REGION Network 36: Interface Signals 06 / Interface Signals ET200SP_204
   // Aufruf des Schnittstellen Signal Bausteins / Call the interface signals bool blocks
   RUNG wire#powerrail
      #instSignalsLeft[43](signal00 := "ET200SP_204"."SP204.00 Main OP: Emergency stop", signal01 := "ET200SP_204".SPARE1, signal02 := "ET200SP_204".SPARE2, signal03 := "ET200SP_204".SPARE3, signal04 := "ET200SP_204".RESERVED, signal05 := "ET200SP_204".SPARE4, signal06 := "ET200SP_204".SPARE5, signal07 := "ET200SP_204".SPARE6, signal08 :=, signal09 :=, signal10 :=, signal11 :=, signal12 :=, signal13 :=, signal14 :=, signal15 :=, interfaceSignals := #statInterfaceSignalsHmi[43].valueSymbolLeft)
      #instSignalsRight[43](signal00 :=, signal01 :=, signal02 :=, signal03 :=, signal04 :=, signal05 :=, signal06 :=, signal07 :=, signal08 :=, signal09 :=, signal10 :=, signal11 :=, signal12 :=, signal13 :=, signal14 :=, signal15 :=, interfaceSignals := #statInterfaceSignalsHmi[43].valueSymbolRight)
   END_RUNG
   // the same network as SCL:
   #instSignalsLeft[43](signal00 := "ET200SP_204"."SP204.00 Main OP: Emergency stop",   // "LAF_InterfaceSignalsBool"
                        signal01 := "ET200SP_204".SPARE1,
                        signal02 := "ET200SP_204".SPARE2,
                        signal03 := "ET200SP_204".SPARE3,
                        signal04 := "ET200SP_204".RESERVED,
                        signal05 := "ET200SP_204".SPARE4,
                        signal06 := "ET200SP_204".SPARE5,
                        signal07 := "ET200SP_204".SPARE6,
                        interfaceSignals := #statInterfaceSignalsHmi[43].valueSymbolLeft,
                        ENO => #_w1);
   IF #_w1 THEN
       #instSignalsRight[43](interfaceSignals := #statInterfaceSignalsHmi[43].valueSymbolRight);   // "LAF_InterfaceSignalsBool"
   END_IF;
END_REGION

REGION Network 37: Interface Signals 06 / Interface Signals ET200SP_205
   // Aufruf des Schnittstellen Signal Bausteins / Call the interface signals bool blocks
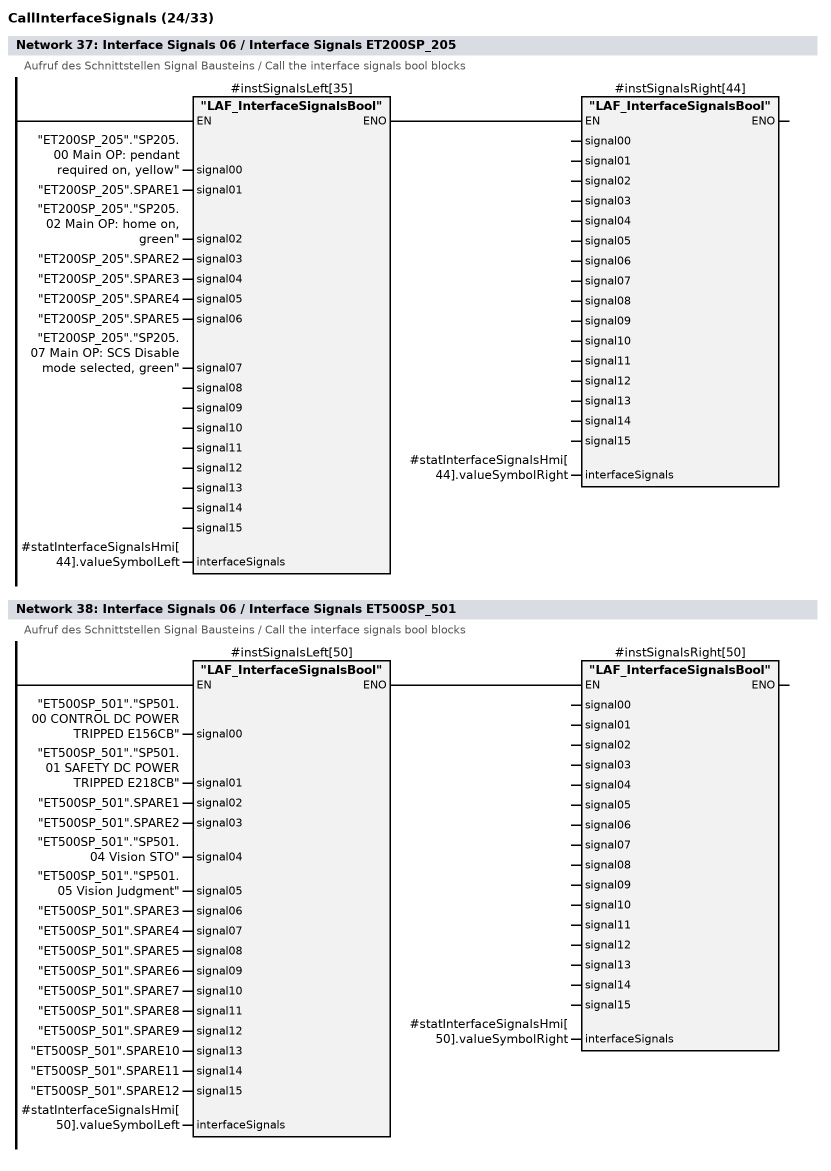
   RUNG wire#powerrail
      #instSignalsLeft[35](signal00 := "ET200SP_205"."SP205.00 Main OP: pendant required on, yellow", signal01 := "ET200SP_205".SPARE1, signal02 := "ET200SP_205"."SP205.02 Main OP: home on, green", signal03 := "ET200SP_205".SPARE2, signal04 := "ET200SP_205".SPARE3, signal05 := "ET200SP_205".SPARE4, signal06 := "ET200SP_205".SPARE5, signal07 := "ET200SP_205"."SP205.07 Main OP: SCS Disable mode selected, green", signal08 :=, signal09 :=, signal10 :=, signal11 :=, signal12 :=, signal13 :=, signal14 :=, signal15 :=, interfaceSignals := #statInterfaceSignalsHmi[44].valueSymbolLeft)
      #instSignalsRight[44](signal00 :=, signal01 :=, signal02 :=, signal03 :=, signal04 :=, signal05 :=, signal06 :=, signal07 :=, signal08 :=, signal09 :=, signal10 :=, signal11 :=, signal12 :=, signal13 :=, signal14 :=, signal15 :=, interfaceSignals := #statInterfaceSignalsHmi[44].valueSymbolRight)
   END_RUNG
   // the same network as SCL:
   #instSignalsLeft[35](signal00 := "ET200SP_205"."SP205.00 Main OP: pendant required on, yellow",   // "LAF_InterfaceSignalsBool"
                        signal01 := "ET200SP_205".SPARE1,
                        signal02 := "ET200SP_205"."SP205.02 Main OP: home on, green",
                        signal03 := "ET200SP_205".SPARE2,
                        signal04 := "ET200SP_205".SPARE3,
                        signal05 := "ET200SP_205".SPARE4,
                        signal06 := "ET200SP_205".SPARE5,
                        signal07 := "ET200SP_205"."SP205.07 Main OP: SCS Disable mode selected, green",
                        interfaceSignals := #statInterfaceSignalsHmi[44].valueSymbolLeft,
                        ENO => #_w1);
   IF #_w1 THEN
       #instSignalsRight[44](interfaceSignals := #statInterfaceSignalsHmi[44].valueSymbolRight);   // "LAF_InterfaceSignalsBool"
   END_IF;
END_REGION

REGION Network 38: Interface Signals 06 / Interface Signals ET500SP_501
   // Aufruf des Schnittstellen Signal Bausteins / Call the interface signals bool blocks
   RUNG wire#powerrail
      #instSignalsLeft[50](signal00 := "ET500SP_501"."SP501.00 CONTROL DC POWER TRIPPED E156CB", signal01 := "ET500SP_501"."SP501.01 SAFETY DC POWER TRIPPED E218CB", signal02 := "ET500SP_501".SPARE1, signal03 := "ET500SP_501".SPARE2, signal04 := "ET500SP_501"."SP501.04 Vision STO", signal05 := "ET500SP_501"."SP501.05 Vision Judgment", signal06 := "ET500SP_501".SPARE3, signal07 := "ET500SP_501".SPARE4, signal08 := "ET500SP_501".SPARE5, signal09 := "ET500SP_501".SPARE6, signal10 := "ET500SP_501".SPARE7, signal11 := "ET500SP_501".SPARE8, signal12 := "ET500SP_501".SPARE9, signal13 := "ET500SP_501".SPARE10, signal14 := "ET500SP_501".SPARE11, signal15 := "ET500SP_501".SPARE12, interfaceSignals := #statInterfaceSignalsHmi[50].valueSymbolLeft)
      #instSignalsRight[50](signal00 :=, signal01 :=, signal02 :=, signal03 :=, signal04 :=, signal05 :=, signal06 :=, signal07 :=, signal08 :=, signal09 :=, signal10 :=, signal11 :=, signal12 :=, signal13 :=, signal14 :=, signal15 :=, interfaceSignals := #statInterfaceSignalsHmi[50].valueSymbolRight)
   END_RUNG
   // the same network as SCL:
   #instSignalsLeft[50](signal00 := "ET500SP_501"."SP501.00 CONTROL DC POWER TRIPPED E156CB",   // "LAF_InterfaceSignalsBool"
                        signal01 := "ET500SP_501"."SP501.01 SAFETY DC POWER TRIPPED E218CB",
                        signal02 := "ET500SP_501".SPARE1,
                        signal03 := "ET500SP_501".SPARE2,
                        signal04 := "ET500SP_501"."SP501.04 Vision STO",
                        signal05 := "ET500SP_501"."SP501.05 Vision Judgment",
                        signal06 := "ET500SP_501".SPARE3,
                        signal07 := "ET500SP_501".SPARE4,
                        signal08 := "ET500SP_501".SPARE5,
                        signal09 := "ET500SP_501".SPARE6,
                        signal10 := "ET500SP_501".SPARE7,
                        signal11 := "ET500SP_501".SPARE8,
                        signal12 := "ET500SP_501".SPARE9,
                        signal13 := "ET500SP_501".SPARE10,
                        signal14 := "ET500SP_501".SPARE11,
                        signal15 := "ET500SP_501".SPARE12,
                        interfaceSignals := #statInterfaceSignalsHmi[50].valueSymbolLeft,
                        ENO => #_w1);
   IF #_w1 THEN
       #instSignalsRight[50](interfaceSignals := #statInterfaceSignalsHmi[50].valueSymbolRight);   // "LAF_InterfaceSignalsBool"
   END_IF;
END_REGION

REGION Network 39: Interface Signals 06 / Interface Signals ET500SP_502
   // Aufruf des Schnittstellen Signal Bausteins / Call the interface signals bool blocks
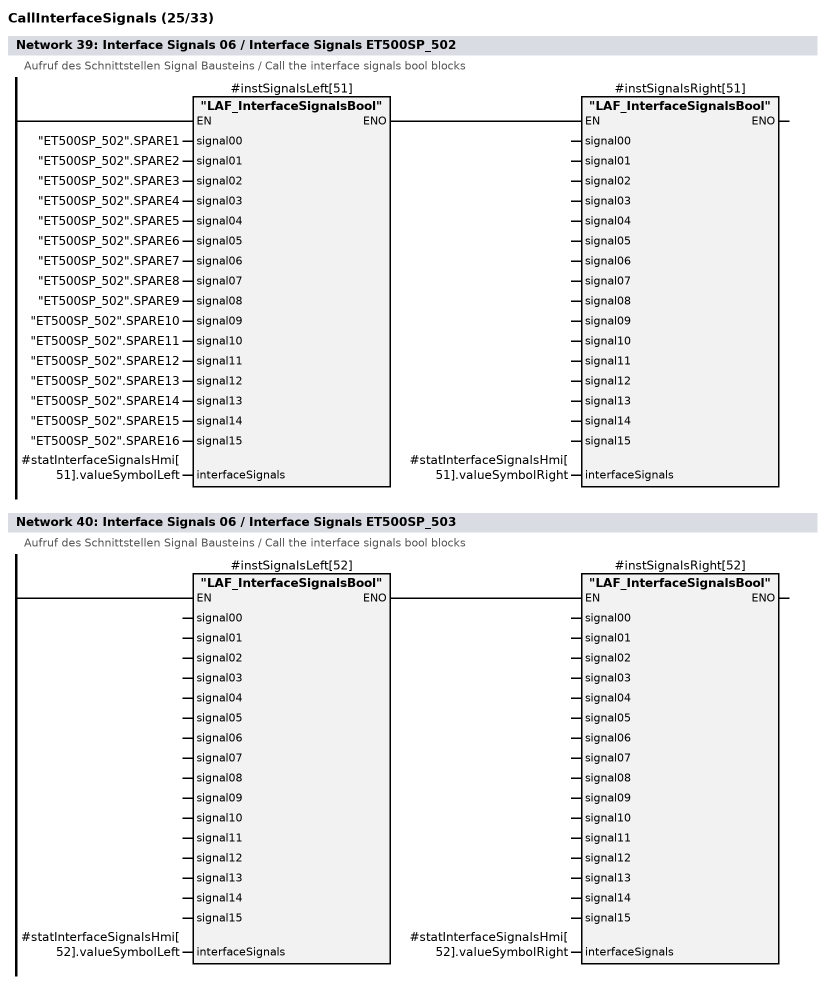
   RUNG wire#powerrail
      #instSignalsLeft[51](signal00 := "ET500SP_502".SPARE1, signal01 := "ET500SP_502".SPARE2, signal02 := "ET500SP_502".SPARE3, signal03 := "ET500SP_502".SPARE4, signal04 := "ET500SP_502".SPARE5, signal05 := "ET500SP_502".SPARE6, signal06 := "ET500SP_502".SPARE7, signal07 := "ET500SP_502".SPARE8, signal08 := "ET500SP_502".SPARE9, signal09 := "ET500SP_502".SPARE10, signal10 := "ET500SP_502".SPARE11, signal11 := "ET500SP_502".SPARE12, signal12 := "ET500SP_502".SPARE13, signal13 := "ET500SP_502".SPARE14, signal14 := "ET500SP_502".SPARE15, signal15 := "ET500SP_502".SPARE16, interfaceSignals := #statInterfaceSignalsHmi[51].valueSymbolLeft)
      #instSignalsRight[51](signal00 :=, signal01 :=, signal02 :=, signal03 :=, signal04 :=, signal05 :=, signal06 :=, signal07 :=, signal08 :=, signal09 :=, signal10 :=, signal11 :=, signal12 :=, signal13 :=, signal14 :=, signal15 :=, interfaceSignals := #statInterfaceSignalsHmi[51].valueSymbolRight)
   END_RUNG
   // the same network as SCL:
   #instSignalsLeft[51](signal00 := "ET500SP_502".SPARE1,   // "LAF_InterfaceSignalsBool"
                        signal01 := "ET500SP_502".SPARE2,
                        signal02 := "ET500SP_502".SPARE3,
                        signal03 := "ET500SP_502".SPARE4,
                        signal04 := "ET500SP_502".SPARE5,
                        signal05 := "ET500SP_502".SPARE6,
                        signal06 := "ET500SP_502".SPARE7,
                        signal07 := "ET500SP_502".SPARE8,
                        signal08 := "ET500SP_502".SPARE9,
                        signal09 := "ET500SP_502".SPARE10,
                        signal10 := "ET500SP_502".SPARE11,
                        signal11 := "ET500SP_502".SPARE12,
                        signal12 := "ET500SP_502".SPARE13,
                        signal13 := "ET500SP_502".SPARE14,
                        signal14 := "ET500SP_502".SPARE15,
                        signal15 := "ET500SP_502".SPARE16,
                        interfaceSignals := #statInterfaceSignalsHmi[51].valueSymbolLeft,
                        ENO => #_w1);
   IF #_w1 THEN
       #instSignalsRight[51](interfaceSignals := #statInterfaceSignalsHmi[51].valueSymbolRight);   // "LAF_InterfaceSignalsBool"
   END_IF;
END_REGION

REGION Network 40: Interface Signals 06 / Interface Signals ET500SP_503
   // Aufruf des Schnittstellen Signal Bausteins / Call the interface signals bool blocks
   RUNG wire#powerrail
      #instSignalsLeft[52](signal00 :=, signal01 :=, signal02 :=, signal03 :=, signal04 :=, signal05 :=, signal06 :=, signal07 :=, signal08 :=, signal09 :=, signal10 :=, signal11 :=, signal12 :=, signal13 :=, signal14 :=, signal15 :=, interfaceSignals := #statInterfaceSignalsHmi[52].valueSymbolLeft)
      #instSignalsRight[52](signal00 :=, signal01 :=, signal02 :=, signal03 :=, signal04 :=, signal05 :=, signal06 :=, signal07 :=, signal08 :=, signal09 :=, signal10 :=, signal11 :=, signal12 :=, signal13 :=, signal14 :=, signal15 :=, interfaceSignals := #statInterfaceSignalsHmi[52].valueSymbolRight)
   END_RUNG
   // the same network as SCL:
   #instSignalsLeft[52](interfaceSignals := #statInterfaceSignalsHmi[52].valueSymbolLeft, ENO => #_w1);   // "LAF_InterfaceSignalsBool"
   IF #_w1 THEN
       #instSignalsRight[52](interfaceSignals := #statInterfaceSignalsHmi[52].valueSymbolRight);   // "LAF_InterfaceSignalsBool"
   END_IF;
END_REGION

REGION Network 41: Interface Signals 06 / Interface Signals ET500SP_504
   // Aufruf des Schnittstellen Signal Bausteins / Call the interface signals bool blocks
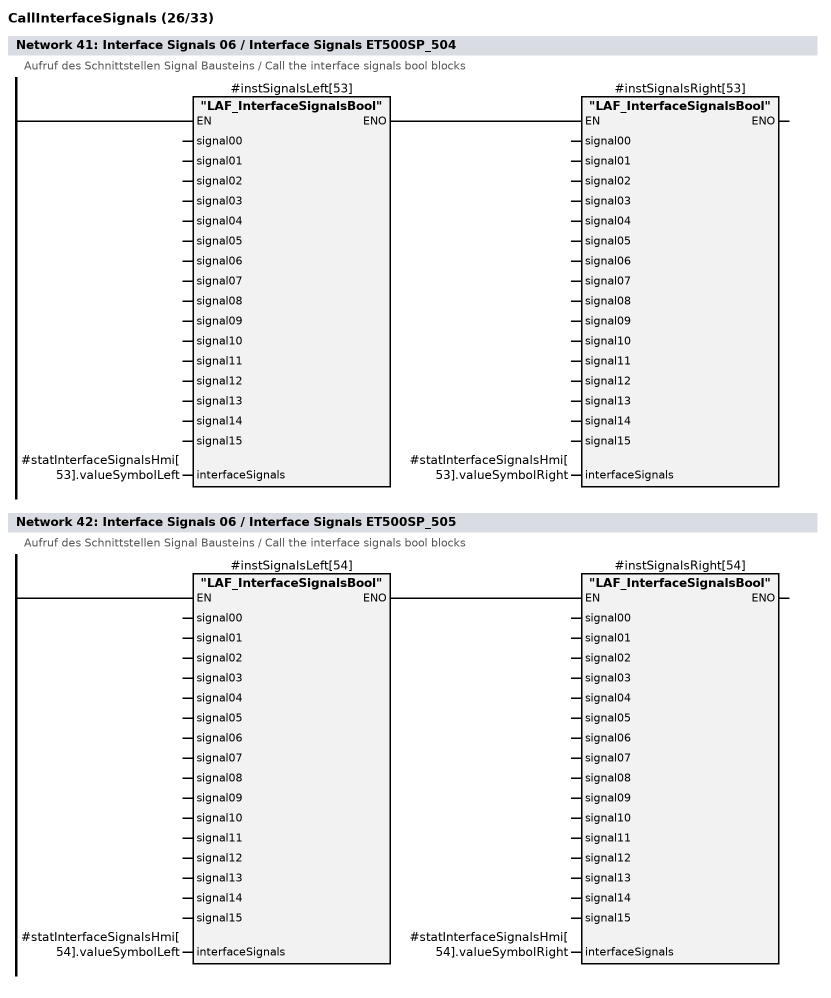
   RUNG wire#powerrail
      #instSignalsLeft[53](signal00 :=, signal01 :=, signal02 :=, signal03 :=, signal04 :=, signal05 :=, signal06 :=, signal07 :=, signal08 :=, signal09 :=, signal10 :=, signal11 :=, signal12 :=, signal13 :=, signal14 :=, signal15 :=, interfaceSignals := #statInterfaceSignalsHmi[53].valueSymbolLeft)
      #instSignalsRight[53](signal00 :=, signal01 :=, signal02 :=, signal03 :=, signal04 :=, signal05 :=, signal06 :=, signal07 :=, signal08 :=, signal09 :=, signal10 :=, signal11 :=, signal12 :=, signal13 :=, signal14 :=, signal15 :=, interfaceSignals := #statInterfaceSignalsHmi[53].valueSymbolRight)
   END_RUNG
   // the same network as SCL:
   #instSignalsLeft[53](interfaceSignals := #statInterfaceSignalsHmi[53].valueSymbolLeft, ENO => #_w1);   // "LAF_InterfaceSignalsBool"
   IF #_w1 THEN
       #instSignalsRight[53](interfaceSignals := #statInterfaceSignalsHmi[53].valueSymbolRight);   // "LAF_InterfaceSignalsBool"
   END_IF;
END_REGION

REGION Network 42: Interface Signals 06 / Interface Signals ET500SP_505
   // Aufruf des Schnittstellen Signal Bausteins / Call the interface signals bool blocks
   RUNG wire#powerrail
      #instSignalsLeft[54](signal00 :=, signal01 :=, signal02 :=, signal03 :=, signal04 :=, signal05 :=, signal06 :=, signal07 :=, signal08 :=, signal09 :=, signal10 :=, signal11 :=, signal12 :=, signal13 :=, signal14 :=, signal15 :=, interfaceSignals := #statInterfaceSignalsHmi[54].valueSymbolLeft)
      #instSignalsRight[54](signal00 :=, signal01 :=, signal02 :=, signal03 :=, signal04 :=, signal05 :=, signal06 :=, signal07 :=, signal08 :=, signal09 :=, signal10 :=, signal11 :=, signal12 :=, signal13 :=, signal14 :=, signal15 :=, interfaceSignals := #statInterfaceSignalsHmi[54].valueSymbolRight)
   END_RUNG
   // the same network as SCL:
   #instSignalsLeft[54](interfaceSignals := #statInterfaceSignalsHmi[54].valueSymbolLeft, ENO => #_w1);   // "LAF_InterfaceSignalsBool"
   IF #_w1 THEN
       #instSignalsRight[54](interfaceSignals := #statInterfaceSignalsHmi[54].valueSymbolRight);   // "LAF_InterfaceSignalsBool"
   END_IF;
END_REGION

REGION Network 43: Interface Signals 06 / Interface Signals ET500SP_506
   // Aufruf des Schnittstellen Signal Bausteins / Call the interface signals bool blocks
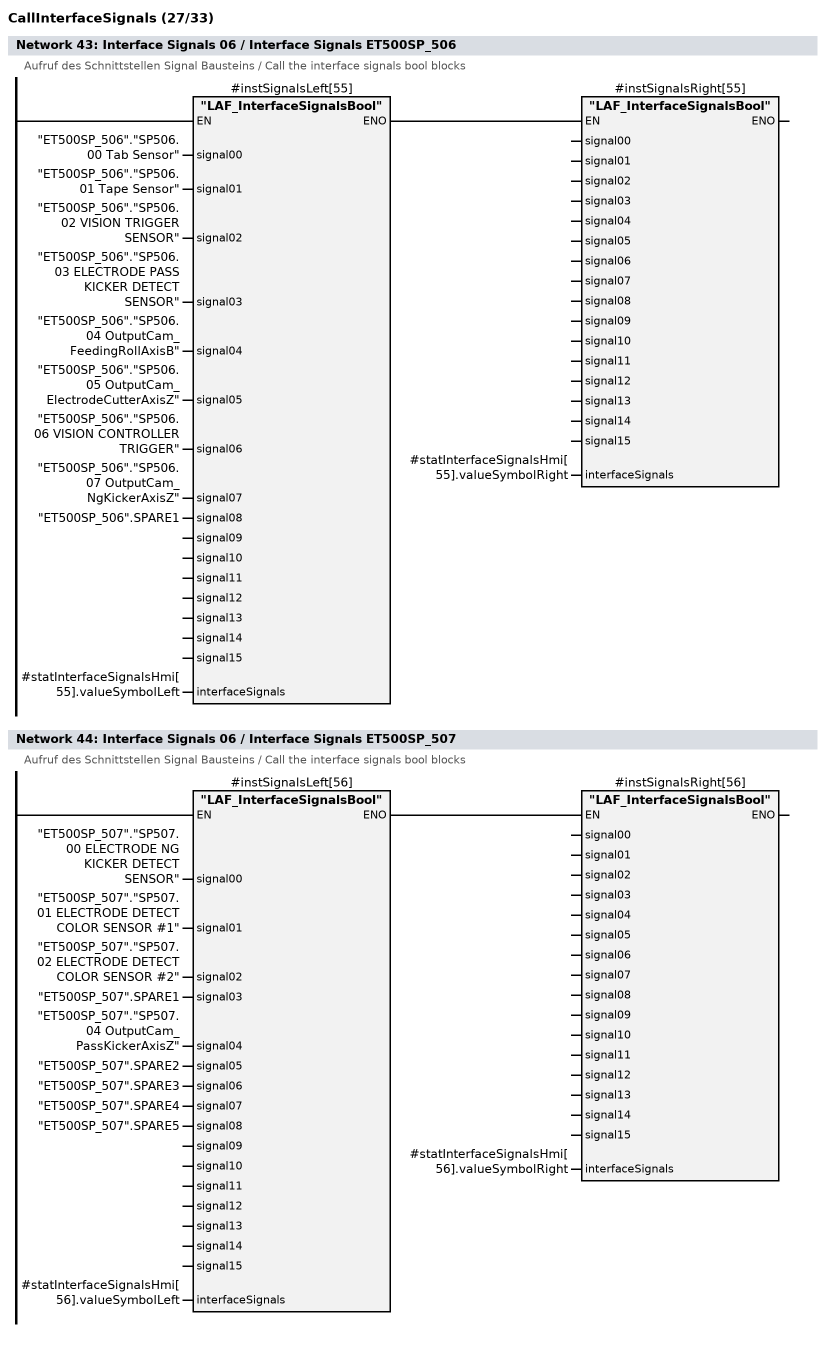
   RUNG wire#powerrail
      #instSignalsLeft[55](signal00 := "ET500SP_506"."SP506.00 Tab Sensor", signal01 := "ET500SP_506"."SP506.01 Tape Sensor", signal02 := "ET500SP_506"."SP506.02 VISION TRIGGER SENSOR", signal03 := "ET500SP_506"."SP506.03 ELECTRODE PASS KICKER DETECT SENSOR", signal04 := "ET500SP_506"."SP506.04 OutputCam_FeedingRollAxisB", signal05 := "ET500SP_506"."SP506.05 OutputCam_ElectrodeCutterAxisZ", signal06 := "ET500SP_506"."SP506.06 VISION CONTROLLER TRIGGER", signal07 := "ET500SP_506"."SP506.07 OutputCam_NgKickerAxisZ", signal08 := "ET500SP_506".SPARE1, signal09 :=, signal10 :=, signal11 :=, signal12 :=, signal13 :=, signal14 :=, signal15 :=, interfaceSignals := #statInterfaceSignalsHmi[55].valueSymbolLeft)
      #instSignalsRight[55](signal00 :=, signal01 :=, signal02 :=, signal03 :=, signal04 :=, signal05 :=, signal06 :=, signal07 :=, signal08 :=, signal09 :=, signal10 :=, signal11 :=, signal12 :=, signal13 :=, signal14 :=, signal15 :=, interfaceSignals := #statInterfaceSignalsHmi[55].valueSymbolRight)
   END_RUNG
   // the same network as SCL:
   #instSignalsLeft[55](signal00 := "ET500SP_506"."SP506.00 Tab Sensor",   // "LAF_InterfaceSignalsBool"
                        signal01 := "ET500SP_506"."SP506.01 Tape Sensor",
                        signal02 := "ET500SP_506"."SP506.02 VISION TRIGGER SENSOR",
                        signal03 := "ET500SP_506"."SP506.03 ELECTRODE PASS KICKER DETECT SENSOR",
                        signal04 := "ET500SP_506"."SP506.04 OutputCam_FeedingRollAxisB",
                        signal05 := "ET500SP_506"."SP506.05 OutputCam_ElectrodeCutterAxisZ",
                        signal06 := "ET500SP_506"."SP506.06 VISION CONTROLLER TRIGGER",
                        signal07 := "ET500SP_506"."SP506.07 OutputCam_NgKickerAxisZ",
                        signal08 := "ET500SP_506".SPARE1,
                        interfaceSignals := #statInterfaceSignalsHmi[55].valueSymbolLeft,
                        ENO => #_w1);
   IF #_w1 THEN
       #instSignalsRight[55](interfaceSignals := #statInterfaceSignalsHmi[55].valueSymbolRight);   // "LAF_InterfaceSignalsBool"
   END_IF;
END_REGION

REGION Network 44: Interface Signals 06 / Interface Signals ET500SP_507
   // Aufruf des Schnittstellen Signal Bausteins / Call the interface signals bool blocks
   RUNG wire#powerrail
      #instSignalsLeft[56](signal00 := "ET500SP_507"."SP507.00 ELECTRODE NG KICKER DETECT SENSOR", signal01 := "ET500SP_507"."SP507.01 ELECTRODE DETECT COLOR SENSOR #1", signal02 := "ET500SP_507"."SP507.02 ELECTRODE DETECT COLOR SENSOR #2", signal03 := "ET500SP_507".SPARE1, signal04 := "ET500SP_507"."SP507.04 OutputCam_PassKickerAxisZ", signal05 := "ET500SP_507".SPARE2, signal06 := "ET500SP_507".SPARE3, signal07 := "ET500SP_507".SPARE4, signal08 := "ET500SP_507".SPARE5, signal09 :=, signal10 :=, signal11 :=, signal12 :=, signal13 :=, signal14 :=, signal15 :=, interfaceSignals := #statInterfaceSignalsHmi[56].valueSymbolLeft)
      #instSignalsRight[56](signal00 :=, signal01 :=, signal02 :=, signal03 :=, signal04 :=, signal05 :=, signal06 :=, signal07 :=, signal08 :=, signal09 :=, signal10 :=, signal11 :=, signal12 :=, signal13 :=, signal14 :=, signal15 :=, interfaceSignals := #statInterfaceSignalsHmi[56].valueSymbolRight)
   END_RUNG
   // the same network as SCL:
   #instSignalsLeft[56](signal00 := "ET500SP_507"."SP507.00 ELECTRODE NG KICKER DETECT SENSOR",   // "LAF_InterfaceSignalsBool"
                        signal01 := "ET500SP_507"."SP507.01 ELECTRODE DETECT COLOR SENSOR #1",
                        signal02 := "ET500SP_507"."SP507.02 ELECTRODE DETECT COLOR SENSOR #2",
                        signal03 := "ET500SP_507".SPARE1,
                        signal04 := "ET500SP_507"."SP507.04 OutputCam_PassKickerAxisZ",
                        signal05 := "ET500SP_507".SPARE2,
                        signal06 := "ET500SP_507".SPARE3,
                        signal07 := "ET500SP_507".SPARE4,
                        signal08 := "ET500SP_507".SPARE5,
                        interfaceSignals := #statInterfaceSignalsHmi[56].valueSymbolLeft,
                        ENO => #_w1);
   IF #_w1 THEN
       #instSignalsRight[56](interfaceSignals := #statInterfaceSignalsHmi[56].valueSymbolRight);   // "LAF_InterfaceSignalsBool"
   END_IF;
END_REGION

REGION Network 45: Interface Signals 06 / Interface Signals ET500SP_508
   // Aufruf des Schnittstellen Signal Bausteins / Call the interface signals bool blocks
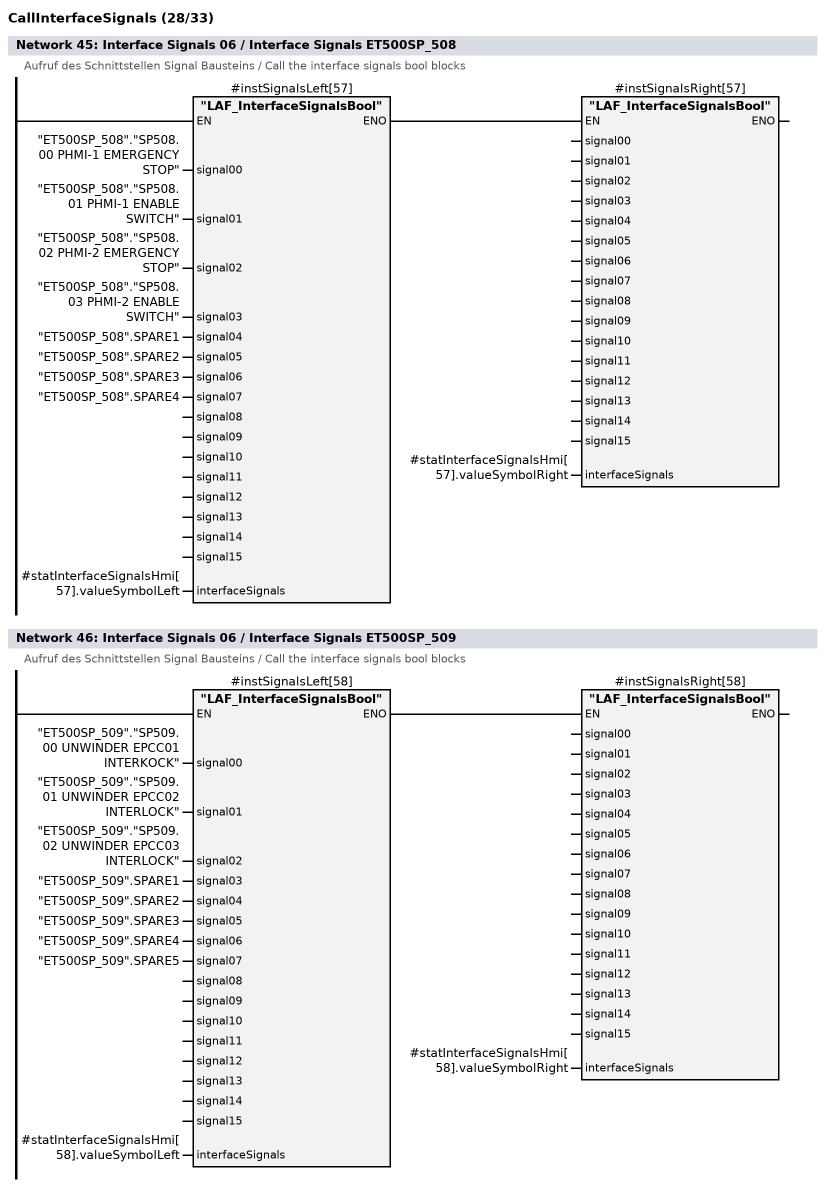
   RUNG wire#powerrail
      #instSignalsLeft[57](signal00 := "ET500SP_508"."SP508.00 PHMI-1 EMERGENCY STOP", signal01 := "ET500SP_508"."SP508.01 PHMI-1 ENABLE SWITCH", signal02 := "ET500SP_508"."SP508.02 PHMI-2 EMERGENCY STOP", signal03 := "ET500SP_508"."SP508.03 PHMI-2 ENABLE SWITCH", signal04 := "ET500SP_508".SPARE1, signal05 := "ET500SP_508".SPARE2, signal06 := "ET500SP_508".SPARE3, signal07 := "ET500SP_508".SPARE4, signal08 :=, signal09 :=, signal10 :=, signal11 :=, signal12 :=, signal13 :=, signal14 :=, signal15 :=, interfaceSignals := #statInterfaceSignalsHmi[57].valueSymbolLeft)
      #instSignalsRight[57](signal00 :=, signal01 :=, signal02 :=, signal03 :=, signal04 :=, signal05 :=, signal06 :=, signal07 :=, signal08 :=, signal09 :=, signal10 :=, signal11 :=, signal12 :=, signal13 :=, signal14 :=, signal15 :=, interfaceSignals := #statInterfaceSignalsHmi[57].valueSymbolRight)
   END_RUNG
   // the same network as SCL:
   #instSignalsLeft[57](signal00 := "ET500SP_508"."SP508.00 PHMI-1 EMERGENCY STOP",   // "LAF_InterfaceSignalsBool"
                        signal01 := "ET500SP_508"."SP508.01 PHMI-1 ENABLE SWITCH",
                        signal02 := "ET500SP_508"."SP508.02 PHMI-2 EMERGENCY STOP",
                        signal03 := "ET500SP_508"."SP508.03 PHMI-2 ENABLE SWITCH",
                        signal04 := "ET500SP_508".SPARE1,
                        signal05 := "ET500SP_508".SPARE2,
                        signal06 := "ET500SP_508".SPARE3,
                        signal07 := "ET500SP_508".SPARE4,
                        interfaceSignals := #statInterfaceSignalsHmi[57].valueSymbolLeft,
                        ENO => #_w1);
   IF #_w1 THEN
       #instSignalsRight[57](interfaceSignals := #statInterfaceSignalsHmi[57].valueSymbolRight);   // "LAF_InterfaceSignalsBool"
   END_IF;
END_REGION

REGION Network 46: Interface Signals 06 / Interface Signals ET500SP_509
   // Aufruf des Schnittstellen Signal Bausteins / Call the interface signals bool blocks
   RUNG wire#powerrail
      #instSignalsLeft[58](signal00 := "ET500SP_509"."SP509.00 UNWINDER EPCC01 INTERKOCK", signal01 := "ET500SP_509"."SP509.01 UNWINDER EPCC02 INTERLOCK", signal02 := "ET500SP_509"."SP509.02 UNWINDER EPCC03 INTERLOCK", signal03 := "ET500SP_509".SPARE1, signal04 := "ET500SP_509".SPARE2, signal05 := "ET500SP_509".SPARE3, signal06 := "ET500SP_509".SPARE4, signal07 := "ET500SP_509".SPARE5, signal08 :=, signal09 :=, signal10 :=, signal11 :=, signal12 :=, signal13 :=, signal14 :=, signal15 :=, interfaceSignals := #statInterfaceSignalsHmi[58].valueSymbolLeft)
      #instSignalsRight[58](signal00 :=, signal01 :=, signal02 :=, signal03 :=, signal04 :=, signal05 :=, signal06 :=, signal07 :=, signal08 :=, signal09 :=, signal10 :=, signal11 :=, signal12 :=, signal13 :=, signal14 :=, signal15 :=, interfaceSignals := #statInterfaceSignalsHmi[58].valueSymbolRight)
   END_RUNG
   // the same network as SCL:
   #instSignalsLeft[58](signal00 := "ET500SP_509"."SP509.00 UNWINDER EPCC01 INTERKOCK",   // "LAF_InterfaceSignalsBool"
                        signal01 := "ET500SP_509"."SP509.01 UNWINDER EPCC02 INTERLOCK",
                        signal02 := "ET500SP_509"."SP509.02 UNWINDER EPCC03 INTERLOCK",
                        signal03 := "ET500SP_509".SPARE1,
                        signal04 := "ET500SP_509".SPARE2,
                        signal05 := "ET500SP_509".SPARE3,
                        signal06 := "ET500SP_509".SPARE4,
                        signal07 := "ET500SP_509".SPARE5,
                        interfaceSignals := #statInterfaceSignalsHmi[58].valueSymbolLeft,
                        ENO => #_w1);
   IF #_w1 THEN
       #instSignalsRight[58](interfaceSignals := #statInterfaceSignalsHmi[58].valueSymbolRight);   // "LAF_InterfaceSignalsBool"
   END_IF;
END_REGION

REGION Network 47: Interface Signals 06 / Interface Signals ET500SP_513
   // Aufruf des Schnittstellen Signal Bausteins / Call the interface signals bool blocks
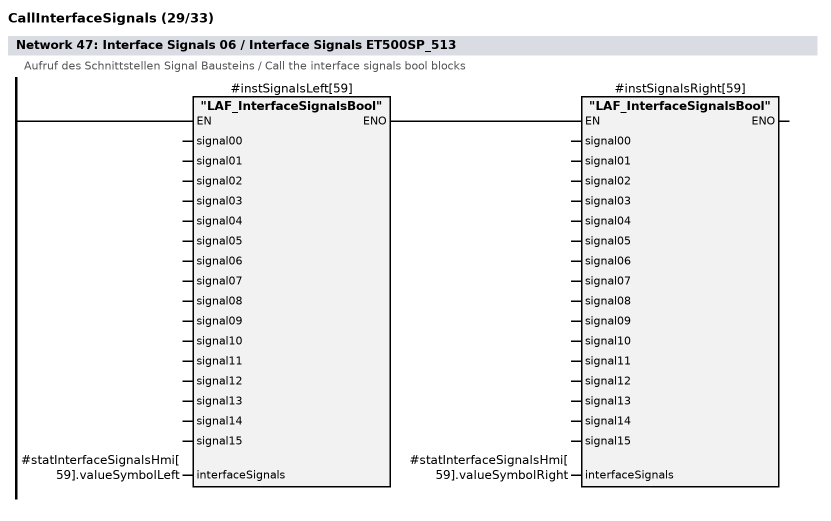
   RUNG wire#powerrail
      #instSignalsLeft[59](signal00 :=, signal01 :=, signal02 :=, signal03 :=, signal04 :=, signal05 :=, signal06 :=, signal07 :=, signal08 :=, signal09 :=, signal10 :=, signal11 :=, signal12 :=, signal13 :=, signal14 :=, signal15 :=, interfaceSignals := #statInterfaceSignalsHmi[59].valueSymbolLeft)
      #instSignalsRight[59](signal00 :=, signal01 :=, signal02 :=, signal03 :=, signal04 :=, signal05 :=, signal06 :=, signal07 :=, signal08 :=, signal09 :=, signal10 :=, signal11 :=, signal12 :=, signal13 :=, signal14 :=, signal15 :=, interfaceSignals := #statInterfaceSignalsHmi[59].valueSymbolRight)
   END_RUNG
   // the same network as SCL:
   #instSignalsLeft[59](interfaceSignals := #statInterfaceSignalsHmi[59].valueSymbolLeft, ENO => #_w1);   // "LAF_InterfaceSignalsBool"
   IF #_w1 THEN
       #instSignalsRight[59](interfaceSignals := #statInterfaceSignalsHmi[59].valueSymbolRight);   // "LAF_InterfaceSignalsBool"
   END_IF;
END_REGION

REGION Network 48: Interface Signals 06 / Interface Signals CPU DI1
   // Aufruf des Schnittstellen Signal Bausteins / Call the interface signals bool blocks
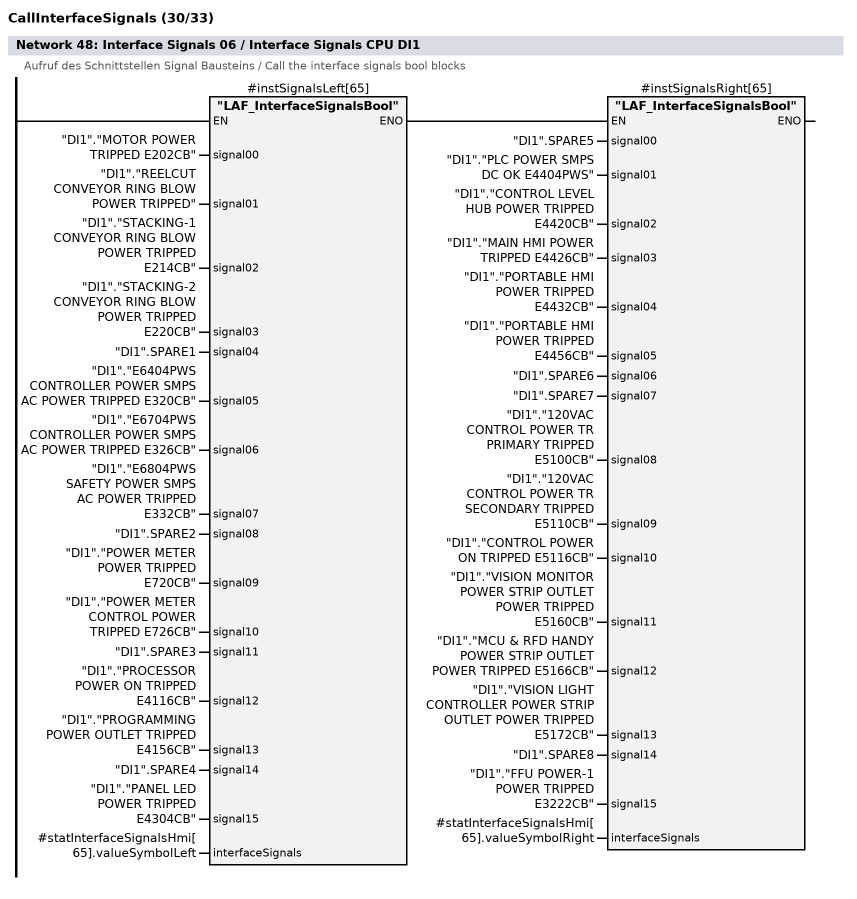
   RUNG wire#powerrail
      #instSignalsLeft[65](signal00 := "DI1"."MOTOR POWER TRIPPED E202CB", signal01 := "DI1"."REELCUT CONVEYOR RING BLOW POWER TRIPPED", signal02 := "DI1"."STACKING-1 CONVEYOR RING BLOW POWER TRIPPED E214CB", signal03 := "DI1"."STACKING-2 CONVEYOR RING BLOW POWER TRIPPED E220CB", signal04 := "DI1".SPARE1, signal05 := "DI1"."E6404PWS CONTROLLER POWER SMPS AC POWER TRIPPED E320CB", signal06 := "DI1"."E6704PWS CONTROLLER POWER SMPS AC POWER TRIPPED E326CB", signal07 := "DI1"."E6804PWS SAFETY POWER SMPS AC POWER TRIPPED E332CB", signal08 := "DI1".SPARE2, signal09 := "DI1"."POWER METER POWER TRIPPED E720CB", signal10 := "DI1"."POWER METER CONTROL POWER TRIPPED E726CB", signal11 := "DI1".SPARE3, signal12 := "DI1"."PROCESSOR POWER ON TRIPPED E4116CB", signal13 := "DI1"."PROGRAMMING POWER OUTLET TRIPPED E4156CB", signal14 := "DI1".SPARE4, signal15 := "DI1"."PANEL LED POWER TRIPPED E4304CB", interfaceSignals := #statInterfaceSignalsHmi[65].valueSymbolLeft)
      #instSignalsRight[65](signal00 := "DI1".SPARE5, signal01 := "DI1"."PLC POWER SMPS DC OK E4404PWS", signal02 := "DI1"."CONTROL LEVEL HUB POWER TRIPPED E4420CB", signal03 := "DI1"."MAIN HMI POWER TRIPPED E4426CB", signal04 := "DI1"."PORTABLE HMI POWER TRIPPED E4432CB", signal05 := "DI1"."PORTABLE HMI POWER TRIPPED E4456CB", signal06 := "DI1".SPARE6, signal07 := "DI1".SPARE7, signal08 := "DI1"."120VAC CONTROL POWER TR PRIMARY TRIPPED E5100CB", signal09 := "DI1"."120VAC CONTROL POWER TR SECONDARY TRIPPED E5110CB", signal10 := "DI1"."CONTROL POWER ON TRIPPED E5116CB", signal11 := "DI1"."VISION MONITOR POWER STRIP OUTLET POWER TRIPPED E5160CB", signal12 := "DI1"."MCU & RFD HANDY POWER STRIP OUTLET POWER TRIPPED E5166CB", signal13 := "DI1"."VISION LIGHT CONTROLLER POWER STRIP OUTLET POWER TRIPPED E5172CB", signal14 := "DI1".SPARE8, signal15 := "DI1"."FFU POWER-1 POWER TRIPPED E3222CB", interfaceSignals := #statInterfaceSignalsHmi[65].valueSymbolRight)
   END_RUNG
   // the same network as SCL:
   #instSignalsLeft[65](signal00 := "DI1"."MOTOR POWER TRIPPED E202CB",   // "LAF_InterfaceSignalsBool"
                        signal01 := "DI1"."REELCUT CONVEYOR RING BLOW POWER TRIPPED",
                        signal02 := "DI1"."STACKING-1 CONVEYOR RING BLOW POWER TRIPPED E214CB",
                        signal03 := "DI1"."STACKING-2 CONVEYOR RING BLOW POWER TRIPPED E220CB",
                        signal04 := "DI1".SPARE1,
                        signal05 := "DI1"."E6404PWS CONTROLLER POWER SMPS AC POWER TRIPPED E320CB",
                        signal06 := "DI1"."E6704PWS CONTROLLER POWER SMPS AC POWER TRIPPED E326CB",
                        signal07 := "DI1"."E6804PWS SAFETY POWER SMPS AC POWER TRIPPED E332CB",
                        signal08 := "DI1".SPARE2,
                        signal09 := "DI1"."POWER METER POWER TRIPPED E720CB",
                        signal10 := "DI1"."POWER METER CONTROL POWER TRIPPED E726CB",
                        signal11 := "DI1".SPARE3,
                        signal12 := "DI1"."PROCESSOR POWER ON TRIPPED E4116CB",
                        signal13 := "DI1"."PROGRAMMING POWER OUTLET TRIPPED E4156CB",
                        signal14 := "DI1".SPARE4,
                        signal15 := "DI1"."PANEL LED POWER TRIPPED E4304CB",
                        interfaceSignals := #statInterfaceSignalsHmi[65].valueSymbolLeft,
                        ENO => #_w1);
   IF #_w1 THEN
       #instSignalsRight[65](signal00 := "DI1".SPARE5,   // "LAF_InterfaceSignalsBool"
                             signal01 := "DI1"."PLC POWER SMPS DC OK E4404PWS",
                             signal02 := "DI1"."CONTROL LEVEL HUB POWER TRIPPED E4420CB",
                             signal03 := "DI1"."MAIN HMI POWER TRIPPED E4426CB",
                             signal04 := "DI1"."PORTABLE HMI POWER TRIPPED E4432CB",
                             signal05 := "DI1"."PORTABLE HMI POWER TRIPPED E4456CB",
                             signal06 := "DI1".SPARE6,
                             signal07 := "DI1".SPARE7,
                             signal08 := "DI1"."120VAC CONTROL POWER TR PRIMARY TRIPPED E5100CB",
                             signal09 := "DI1"."120VAC CONTROL POWER TR SECONDARY TRIPPED E5110CB",
                             signal10 := "DI1"."CONTROL POWER ON TRIPPED E5116CB",
                             signal11 := "DI1"."VISION MONITOR POWER STRIP OUTLET POWER TRIPPED E5160CB",
                             signal12 := "DI1"."MCU & RFD HANDY POWER STRIP OUTLET POWER TRIPPED E5166CB",
                             signal13 := "DI1"."VISION LIGHT CONTROLLER POWER STRIP OUTLET POWER TRIPPED E5172CB",
                             signal14 := "DI1".SPARE8,
                             signal15 := "DI1"."FFU POWER-1 POWER TRIPPED E3222CB",
                             interfaceSignals := #statInterfaceSignalsHmi[65].valueSymbolRight);
   END_IF;
END_REGION

REGION Network 49: Interface Signals 06 / Interface Signals CPU DI2
   // Aufruf des Schnittstellen Signal Bausteins / Call the interface signals bool blocks
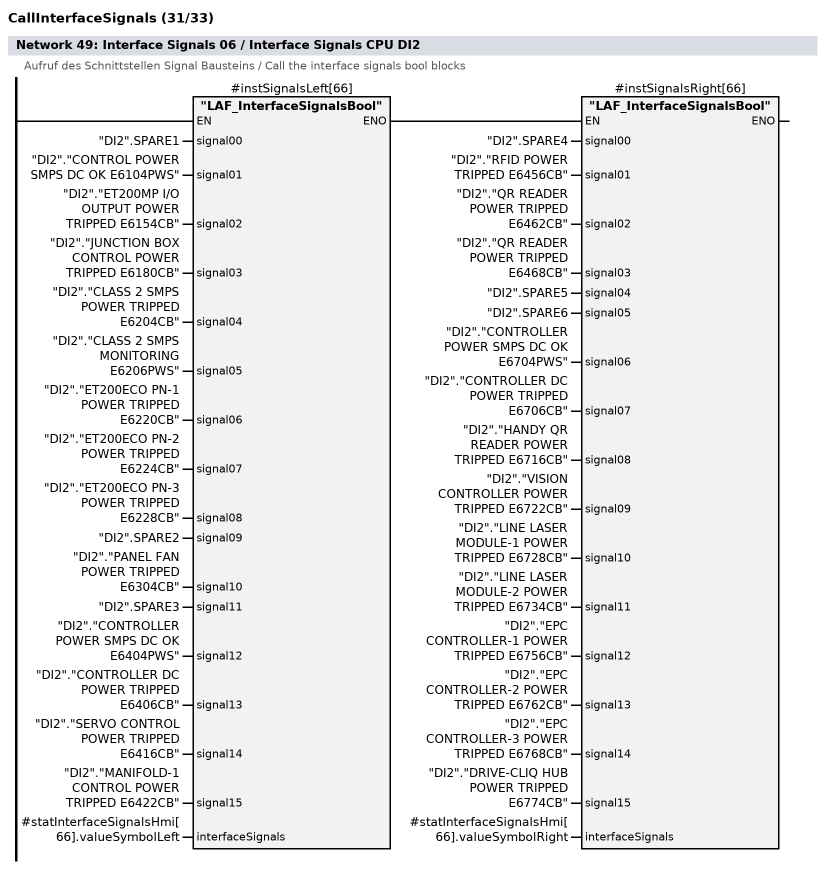
   RUNG wire#powerrail
      #instSignalsLeft[66](signal00 := "DI2".SPARE1, signal01 := "DI2"."CONTROL POWER SMPS DC OK E6104PWS", signal02 := "DI2"."ET200MP I/O OUTPUT POWER TRIPPED E6154CB", signal03 := "DI2"."JUNCTION BOX CONTROL POWER TRIPPED E6180CB", signal04 := "DI2"."CLASS 2 SMPS POWER TRIPPED E6204CB", signal05 := "DI2"."CLASS 2 SMPS MONITORING E6206PWS", signal06 := "DI2"."ET200ECO PN-1 POWER TRIPPED E6220CB", signal07 := "DI2"."ET200ECO PN-2 POWER TRIPPED E6224CB", signal08 := "DI2"."ET200ECO PN-3 POWER TRIPPED E6228CB", signal09 := "DI2".SPARE2, signal10 := "DI2"."PANEL FAN POWER TRIPPED E6304CB", signal11 := "DI2".SPARE3, signal12 := "DI2"."CONTROLLER POWER SMPS DC OK E6404PWS", signal13 := "DI2"."CONTROLLER DC POWER TRIPPED E6406CB", signal14 := "DI2"."SERVO CONTROL POWER TRIPPED E6416CB", signal15 := "DI2"."MANIFOLD-1 CONTROL POWER TRIPPED E6422CB", interfaceSignals := #statInterfaceSignalsHmi[66].valueSymbolLeft)
      #instSignalsRight[66](signal00 := "DI2".SPARE4, signal01 := "DI2"."RFID POWER TRIPPED E6456CB", signal02 := "DI2"."QR READER POWER TRIPPED E6462CB", signal03 := "DI2"."QR READER POWER TRIPPED E6468CB", signal04 := "DI2".SPARE5, signal05 := "DI2".SPARE6, signal06 := "DI2"."CONTROLLER POWER SMPS DC OK E6704PWS", signal07 := "DI2"."CONTROLLER DC POWER TRIPPED E6706CB", signal08 := "DI2"."HANDY QR READER POWER TRIPPED E6716CB", signal09 := "DI2"."VISION CONTROLLER POWER TRIPPED E6722CB", signal10 := "DI2"."LINE LASER MODULE-1 POWER TRIPPED E6728CB", signal11 := "DI2"."LINE LASER MODULE-2 POWER TRIPPED E6734CB", signal12 := "DI2"."EPC CONTROLLER-1 POWER TRIPPED E6756CB", signal13 := "DI2"."EPC CONTROLLER-2 POWER TRIPPED E6762CB", signal14 := "DI2"."EPC CONTROLLER-3 POWER TRIPPED E6768CB", signal15 := "DI2"."DRIVE-CLIQ HUB POWER TRIPPED E6774CB", interfaceSignals := #statInterfaceSignalsHmi[66].valueSymbolRight)
   END_RUNG
   // the same network as SCL:
   #instSignalsLeft[66](signal00 := "DI2".SPARE1,   // "LAF_InterfaceSignalsBool"
                        signal01 := "DI2"."CONTROL POWER SMPS DC OK E6104PWS",
                        signal02 := "DI2"."ET200MP I/O OUTPUT POWER TRIPPED E6154CB",
                        signal03 := "DI2"."JUNCTION BOX CONTROL POWER TRIPPED E6180CB",
                        signal04 := "DI2"."CLASS 2 SMPS POWER TRIPPED E6204CB",
                        signal05 := "DI2"."CLASS 2 SMPS MONITORING E6206PWS",
                        signal06 := "DI2"."ET200ECO PN-1 POWER TRIPPED E6220CB",
                        signal07 := "DI2"."ET200ECO PN-2 POWER TRIPPED E6224CB",
                        signal08 := "DI2"."ET200ECO PN-3 POWER TRIPPED E6228CB",
                        signal09 := "DI2".SPARE2,
                        signal10 := "DI2"."PANEL FAN POWER TRIPPED E6304CB",
                        signal11 := "DI2".SPARE3,
                        signal12 := "DI2"."CONTROLLER POWER SMPS DC OK E6404PWS",
                        signal13 := "DI2"."CONTROLLER DC POWER TRIPPED E6406CB",
                        signal14 := "DI2"."SERVO CONTROL POWER TRIPPED E6416CB",
                        signal15 := "DI2"."MANIFOLD-1 CONTROL POWER TRIPPED E6422CB",
                        interfaceSignals := #statInterfaceSignalsHmi[66].valueSymbolLeft,
                        ENO => #_w1);
   IF #_w1 THEN
       #instSignalsRight[66](signal00 := "DI2".SPARE4,   // "LAF_InterfaceSignalsBool"
                             signal01 := "DI2"."RFID POWER TRIPPED E6456CB",
                             signal02 := "DI2"."QR READER POWER TRIPPED E6462CB",
                             signal03 := "DI2"."QR READER POWER TRIPPED E6468CB",
                             signal04 := "DI2".SPARE5,
                             signal05 := "DI2".SPARE6,
                             signal06 := "DI2"."CONTROLLER POWER SMPS DC OK E6704PWS",
                             signal07 := "DI2"."CONTROLLER DC POWER TRIPPED E6706CB",
                             signal08 := "DI2"."HANDY QR READER POWER TRIPPED E6716CB",
                             signal09 := "DI2"."VISION CONTROLLER POWER TRIPPED E6722CB",
                             signal10 := "DI2"."LINE LASER MODULE-1 POWER TRIPPED E6728CB",
                             signal11 := "DI2"."LINE LASER MODULE-2 POWER TRIPPED E6734CB",
                             signal12 := "DI2"."EPC CONTROLLER-1 POWER TRIPPED E6756CB",
                             signal13 := "DI2"."EPC CONTROLLER-2 POWER TRIPPED E6762CB",
                             signal14 := "DI2"."EPC CONTROLLER-3 POWER TRIPPED E6768CB",
                             signal15 := "DI2"."DRIVE-CLIQ HUB POWER TRIPPED E6774CB",
                             interfaceSignals := #statInterfaceSignalsHmi[66].valueSymbolRight);
   END_IF;
END_REGION

REGION Network 50: Interface Signals 06 / Interface Signals CPU DI3
   // Aufruf des Schnittstellen Signal Bausteins / Call the interface signals bool blocks
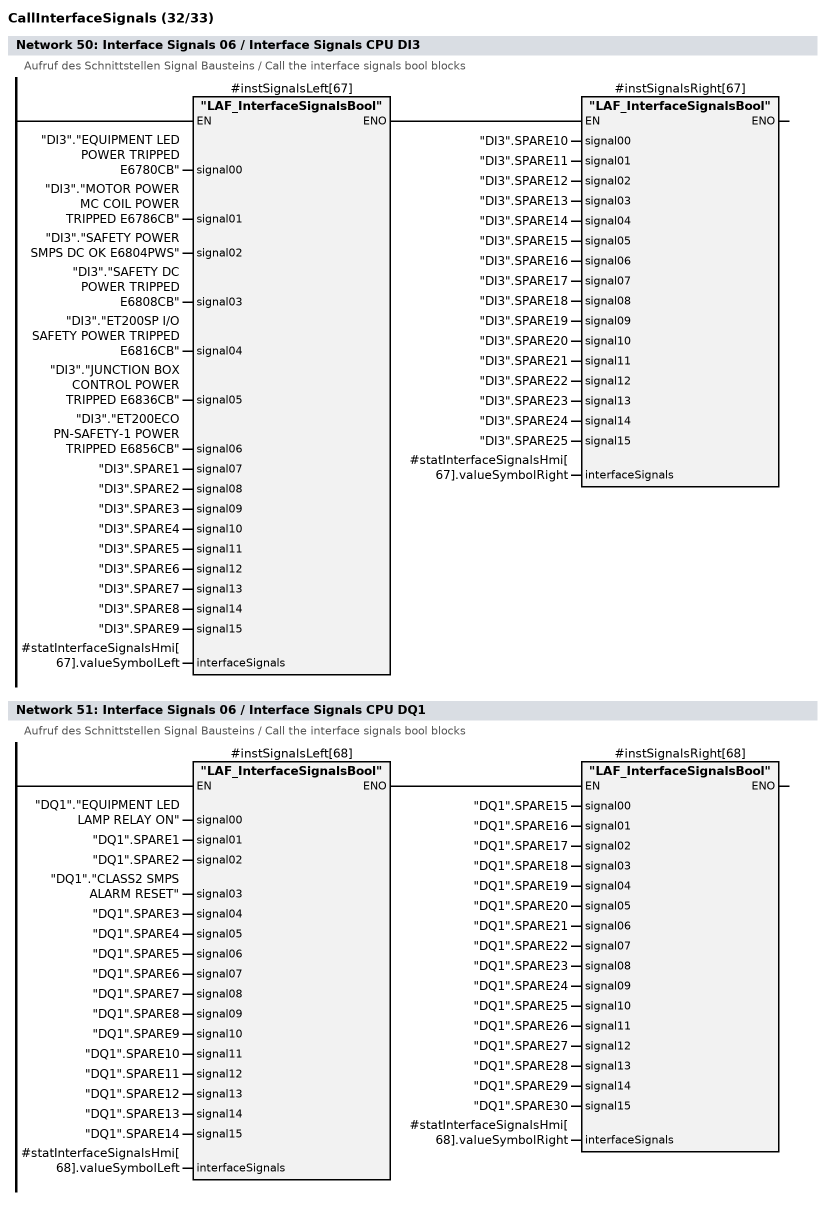
   RUNG wire#powerrail
      #instSignalsLeft[67](signal00 := "DI3"."EQUIPMENT LED POWER TRIPPED E6780CB", signal01 := "DI3"."MOTOR POWER MC COIL POWER TRIPPED E6786CB", signal02 := "DI3"."SAFETY POWER SMPS DC OK E6804PWS", signal03 := "DI3"."SAFETY DC POWER TRIPPED E6808CB", signal04 := "DI3"."ET200SP I/O SAFETY POWER TRIPPED E6816CB", signal05 := "DI3"."JUNCTION BOX CONTROL POWER TRIPPED E6836CB", signal06 := "DI3"."ET200ECO PN-SAFETY-1 POWER TRIPPED E6856CB", signal07 := "DI3".SPARE1, signal08 := "DI3".SPARE2, signal09 := "DI3".SPARE3, signal10 := "DI3".SPARE4, signal11 := "DI3".SPARE5, signal12 := "DI3".SPARE6, signal13 := "DI3".SPARE7, signal14 := "DI3".SPARE8, signal15 := "DI3".SPARE9, interfaceSignals := #statInterfaceSignalsHmi[67].valueSymbolLeft)
      #instSignalsRight[67](signal00 := "DI3".SPARE10, signal01 := "DI3".SPARE11, signal02 := "DI3".SPARE12, signal03 := "DI3".SPARE13, signal04 := "DI3".SPARE14, signal05 := "DI3".SPARE15, signal06 := "DI3".SPARE16, signal07 := "DI3".SPARE17, signal08 := "DI3".SPARE18, signal09 := "DI3".SPARE19, signal10 := "DI3".SPARE20, signal11 := "DI3".SPARE21, signal12 := "DI3".SPARE22, signal13 := "DI3".SPARE23, signal14 := "DI3".SPARE24, signal15 := "DI3".SPARE25, interfaceSignals := #statInterfaceSignalsHmi[67].valueSymbolRight)
   END_RUNG
   // the same network as SCL:
   #instSignalsLeft[67](signal00 := "DI3"."EQUIPMENT LED POWER TRIPPED E6780CB",   // "LAF_InterfaceSignalsBool"
                        signal01 := "DI3"."MOTOR POWER MC COIL POWER TRIPPED E6786CB",
                        signal02 := "DI3"."SAFETY POWER SMPS DC OK E6804PWS",
                        signal03 := "DI3"."SAFETY DC POWER TRIPPED E6808CB",
                        signal04 := "DI3"."ET200SP I/O SAFETY POWER TRIPPED E6816CB",
                        signal05 := "DI3"."JUNCTION BOX CONTROL POWER TRIPPED E6836CB",
                        signal06 := "DI3"."ET200ECO PN-SAFETY-1 POWER TRIPPED E6856CB",
                        signal07 := "DI3".SPARE1,
                        signal08 := "DI3".SPARE2,
                        signal09 := "DI3".SPARE3,
                        signal10 := "DI3".SPARE4,
                        signal11 := "DI3".SPARE5,
                        signal12 := "DI3".SPARE6,
                        signal13 := "DI3".SPARE7,
                        signal14 := "DI3".SPARE8,
                        signal15 := "DI3".SPARE9,
                        interfaceSignals := #statInterfaceSignalsHmi[67].valueSymbolLeft,
                        ENO => #_w1);
   IF #_w1 THEN
       #instSignalsRight[67](signal00 := "DI3".SPARE10,   // "LAF_InterfaceSignalsBool"
                             signal01 := "DI3".SPARE11,
                             signal02 := "DI3".SPARE12,
                             signal03 := "DI3".SPARE13,
                             signal04 := "DI3".SPARE14,
                             signal05 := "DI3".SPARE15,
                             signal06 := "DI3".SPARE16,
                             signal07 := "DI3".SPARE17,
                             signal08 := "DI3".SPARE18,
                             signal09 := "DI3".SPARE19,
                             signal10 := "DI3".SPARE20,
                             signal11 := "DI3".SPARE21,
                             signal12 := "DI3".SPARE22,
                             signal13 := "DI3".SPARE23,
                             signal14 := "DI3".SPARE24,
                             signal15 := "DI3".SPARE25,
                             interfaceSignals := #statInterfaceSignalsHmi[67].valueSymbolRight);
   END_IF;
END_REGION

REGION Network 51: Interface Signals 06 / Interface Signals CPU DQ1
   // Aufruf des Schnittstellen Signal Bausteins / Call the interface signals bool blocks
   RUNG wire#powerrail
      #instSignalsLeft[68](signal00 := "DQ1"."EQUIPMENT LED LAMP RELAY ON", signal01 := "DQ1".SPARE1, signal02 := "DQ1".SPARE2, signal03 := "DQ1"."CLASS2 SMPS ALARM RESET", signal04 := "DQ1".SPARE3, signal05 := "DQ1".SPARE4, signal06 := "DQ1".SPARE5, signal07 := "DQ1".SPARE6, signal08 := "DQ1".SPARE7, signal09 := "DQ1".SPARE8, signal10 := "DQ1".SPARE9, signal11 := "DQ1".SPARE10, signal12 := "DQ1".SPARE11, signal13 := "DQ1".SPARE12, signal14 := "DQ1".SPARE13, signal15 := "DQ1".SPARE14, interfaceSignals := #statInterfaceSignalsHmi[68].valueSymbolLeft)
      #instSignalsRight[68](signal00 := "DQ1".SPARE15, signal01 := "DQ1".SPARE16, signal02 := "DQ1".SPARE17, signal03 := "DQ1".SPARE18, signal04 := "DQ1".SPARE19, signal05 := "DQ1".SPARE20, signal06 := "DQ1".SPARE21, signal07 := "DQ1".SPARE22, signal08 := "DQ1".SPARE23, signal09 := "DQ1".SPARE24, signal10 := "DQ1".SPARE25, signal11 := "DQ1".SPARE26, signal12 := "DQ1".SPARE27, signal13 := "DQ1".SPARE28, signal14 := "DQ1".SPARE29, signal15 := "DQ1".SPARE30, interfaceSignals := #statInterfaceSignalsHmi[68].valueSymbolRight)
   END_RUNG
   // the same network as SCL:
   #instSignalsLeft[68](signal00 := "DQ1"."EQUIPMENT LED LAMP RELAY ON",   // "LAF_InterfaceSignalsBool"
                        signal01 := "DQ1".SPARE1,
                        signal02 := "DQ1".SPARE2,
                        signal03 := "DQ1"."CLASS2 SMPS ALARM RESET",
                        signal04 := "DQ1".SPARE3,
                        signal05 := "DQ1".SPARE4,
                        signal06 := "DQ1".SPARE5,
                        signal07 := "DQ1".SPARE6,
                        signal08 := "DQ1".SPARE7,
                        signal09 := "DQ1".SPARE8,
                        signal10 := "DQ1".SPARE9,
                        signal11 := "DQ1".SPARE10,
                        signal12 := "DQ1".SPARE11,
                        signal13 := "DQ1".SPARE12,
                        signal14 := "DQ1".SPARE13,
                        signal15 := "DQ1".SPARE14,
                        interfaceSignals := #statInterfaceSignalsHmi[68].valueSymbolLeft,
                        ENO => #_w1);
   IF #_w1 THEN
       #instSignalsRight[68](signal00 := "DQ1".SPARE15,   // "LAF_InterfaceSignalsBool"
                             signal01 := "DQ1".SPARE16,
                             signal02 := "DQ1".SPARE17,
                             signal03 := "DQ1".SPARE18,
                             signal04 := "DQ1".SPARE19,
                             signal05 := "DQ1".SPARE20,
                             signal06 := "DQ1".SPARE21,
                             signal07 := "DQ1".SPARE22,
                             signal08 := "DQ1".SPARE23,
                             signal09 := "DQ1".SPARE24,
                             signal10 := "DQ1".SPARE25,
                             signal11 := "DQ1".SPARE26,
                             signal12 := "DQ1".SPARE27,
                             signal13 := "DQ1".SPARE28,
                             signal14 := "DQ1".SPARE29,
                             signal15 := "DQ1".SPARE30,
                             interfaceSignals := #statInterfaceSignalsHmi[68].valueSymbolRight);
   END_IF;
END_REGION

REGION Network 52: Interface Signals 06 / Interface Signals CPU FDI1
   // Aufruf des Schnittstellen Signal Bausteins / Call the interface signals bool blocks
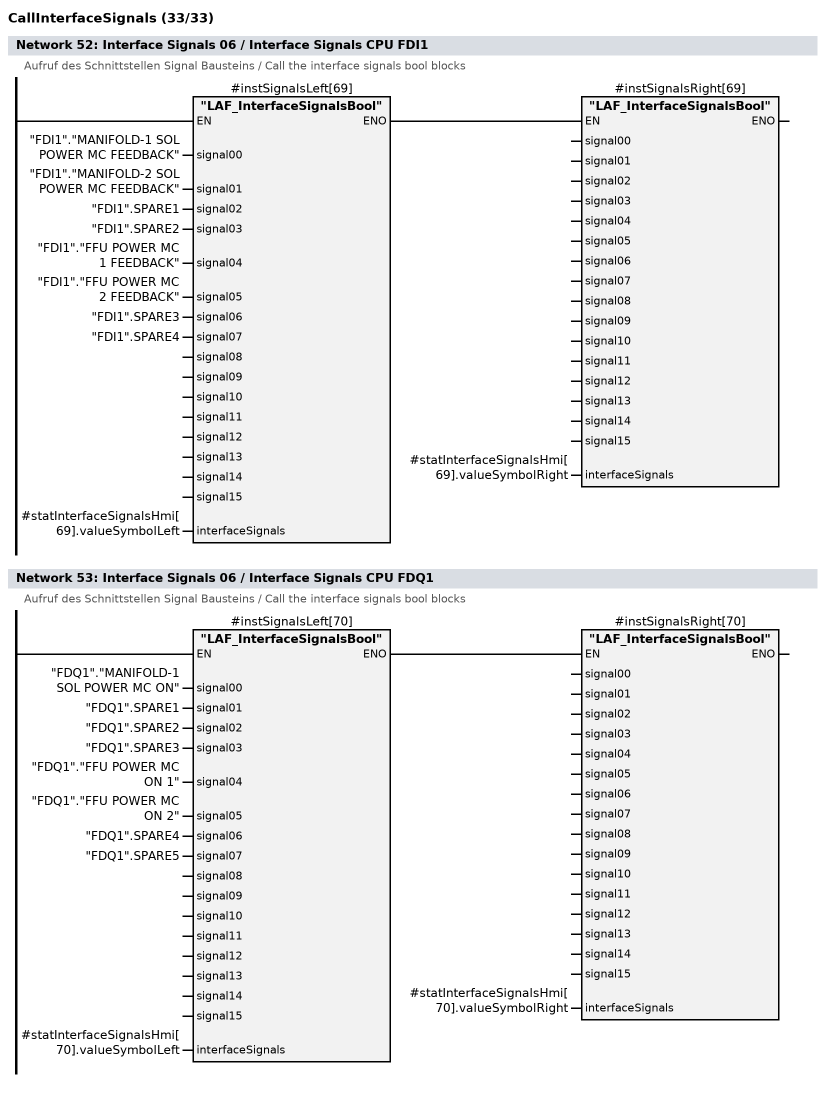
   RUNG wire#powerrail
      #instSignalsLeft[69](signal00 := "FDI1"."MANIFOLD-1 SOL POWER MC FEEDBACK", signal01 := "FDI1"."MANIFOLD-2 SOL POWER MC FEEDBACK", signal02 := "FDI1".SPARE1, signal03 := "FDI1".SPARE2, signal04 := "FDI1"."FFU POWER MC 1 FEEDBACK", signal05 := "FDI1"."FFU POWER MC 2 FEEDBACK", signal06 := "FDI1".SPARE3, signal07 := "FDI1".SPARE4, signal08 :=, signal09 :=, signal10 :=, signal11 :=, signal12 :=, signal13 :=, signal14 :=, signal15 :=, interfaceSignals := #statInterfaceSignalsHmi[69].valueSymbolLeft)
      #instSignalsRight[69](signal00 :=, signal01 :=, signal02 :=, signal03 :=, signal04 :=, signal05 :=, signal06 :=, signal07 :=, signal08 :=, signal09 :=, signal10 :=, signal11 :=, signal12 :=, signal13 :=, signal14 :=, signal15 :=, interfaceSignals := #statInterfaceSignalsHmi[69].valueSymbolRight)
   END_RUNG
   // the same network as SCL:
   #instSignalsLeft[69](signal00 := "FDI1"."MANIFOLD-1 SOL POWER MC FEEDBACK",   // "LAF_InterfaceSignalsBool"
                        signal01 := "FDI1"."MANIFOLD-2 SOL POWER MC FEEDBACK",
                        signal02 := "FDI1".SPARE1,
                        signal03 := "FDI1".SPARE2,
                        signal04 := "FDI1"."FFU POWER MC 1 FEEDBACK",
                        signal05 := "FDI1"."FFU POWER MC 2 FEEDBACK",
                        signal06 := "FDI1".SPARE3,
                        signal07 := "FDI1".SPARE4,
                        interfaceSignals := #statInterfaceSignalsHmi[69].valueSymbolLeft,
                        ENO => #_w1);
   IF #_w1 THEN
       #instSignalsRight[69](interfaceSignals := #statInterfaceSignalsHmi[69].valueSymbolRight);   // "LAF_InterfaceSignalsBool"
   END_IF;
END_REGION

REGION Network 53: Interface Signals 06 / Interface Signals CPU FDQ1
   // Aufruf des Schnittstellen Signal Bausteins / Call the interface signals bool blocks
   RUNG wire#powerrail
      #instSignalsLeft[70](signal00 := "FDQ1"."MANIFOLD-1 SOL POWER MC ON", signal01 := "FDQ1".SPARE1, signal02 := "FDQ1".SPARE2, signal03 := "FDQ1".SPARE3, signal04 := "FDQ1"."FFU POWER MC ON 1", signal05 := "FDQ1"."FFU POWER MC ON 2", signal06 := "FDQ1".SPARE4, signal07 := "FDQ1".SPARE5, signal08 :=, signal09 :=, signal10 :=, signal11 :=, signal12 :=, signal13 :=, signal14 :=, signal15 :=, interfaceSignals := #statInterfaceSignalsHmi[70].valueSymbolLeft)
      #instSignalsRight[70](signal00 :=, signal01 :=, signal02 :=, signal03 :=, signal04 :=, signal05 :=, signal06 :=, signal07 :=, signal08 :=, signal09 :=, signal10 :=, signal11 :=, signal12 :=, signal13 :=, signal14 :=, signal15 :=, interfaceSignals := #statInterfaceSignalsHmi[70].valueSymbolRight)
   END_RUNG
   // the same network as SCL:
   #instSignalsLeft[70](signal00 := "FDQ1"."MANIFOLD-1 SOL POWER MC ON",   // "LAF_InterfaceSignalsBool"
                        signal01 := "FDQ1".SPARE1,
                        signal02 := "FDQ1".SPARE2,
                        signal03 := "FDQ1".SPARE3,
                        signal04 := "FDQ1"."FFU POWER MC ON 1",
                        signal05 := "FDQ1"."FFU POWER MC ON 2",
                        signal06 := "FDQ1".SPARE4,
                        signal07 := "FDQ1".SPARE5,
                        interfaceSignals := #statInterfaceSignalsHmi[70].valueSymbolLeft,
                        ENO => #_w1);
   IF #_w1 THEN
       #instSignalsRight[70](interfaceSignals := #statInterfaceSignalsHmi[70].valueSymbolRight);   // "LAF_InterfaceSignalsBool"
   END_IF;
END_REGION
END_FUNCTION_BLOCK

FUNCTION_BLOCK "CallInterfaceSignalsConv"   // FB97, LAD
// stored: MemoryReserve 100, SetENOAutomatically false
   VAR_INPUT
      InterfaceTestMode : Bool;
   END_VAR
   VAR_OUTPUT
      signalsR2S : "typeReelCutToStack";
      signalsS2R : "typeStackToReelCut";
   END_VAR
   VAR_IN_OUT
      CommR2S : Array[0..95] of Bool;
      CommS2R : Array[0..95] of Bool;
      InterfaceTestButton : "LER_SignalsInput";
   END_VAR
   VAR
      statWordBuffer_1 : Array[0..5] of Word;
      statWordBuffer_2 : Array[0..5] of Word;
   END_VAR
   VAR_TEMP
      tempDeleteData : "LER_SignalsInput";
   END_VAR
   VAR CONSTANT
      TRUE : Bool := TRUE;
   END_VAR
   VAR_TEMP   // added for the SCL form of the ladder/FBD networks
      _w1 : Bool;
      _w2 : Bool;
      _w3 : Bool;
      _w4 : Bool;
   END_VAR
BEGIN

REGION Network 1: CommR2S -> signalsR2S
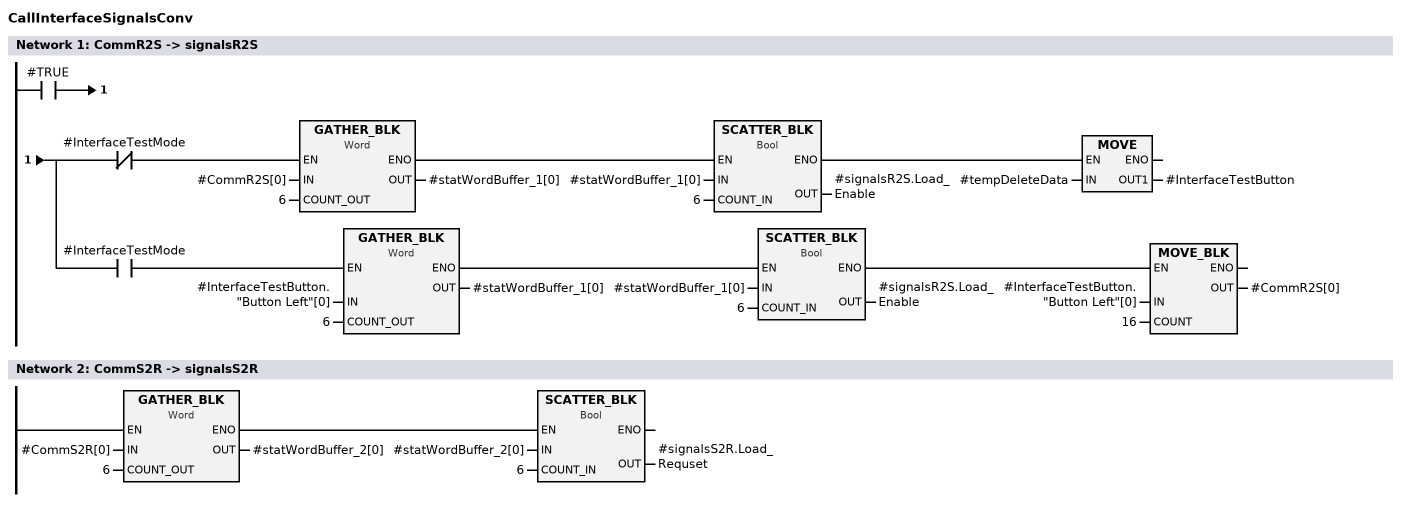
   GATHER_BLK(EN := #TRUE AND NOT #InterfaceTestMode,
              IN := #CommR2S[0],
              COUNT_OUT := 6,
              OUT => #statWordBuffer_1[0],
              ENO => #_w1);
   SCATTER_BLK(EN := #_w1,
               IN := #statWordBuffer_1[0],
               COUNT_IN := 6,
               OUT => #signalsR2S.Load_Enable,
               ENO => #_w2);
   IF #_w2 THEN #InterfaceTestButton := #tempDeleteData; END_IF;
   GATHER_BLK(EN := #TRUE AND #InterfaceTestMode,
              IN := #InterfaceTestButton."Button Left"[0],
              COUNT_OUT := 6,
              OUT => #statWordBuffer_1[0],
              ENO => #_w3);
   SCATTER_BLK(EN := #_w3,
               IN := #statWordBuffer_1[0],
               COUNT_IN := 6,
               OUT => #signalsR2S.Load_Enable,
               ENO => #_w4);
   IF #_w4 THEN
       MOVE_BLK(IN := #InterfaceTestButton."Button Left"[0], COUNT := 16, OUT => #CommR2S[0]);
   END_IF;
END_REGION

REGION Network 2: CommS2R -> signalsS2R
   RUNG wire#powerrail
      { S7_Templates := "[dest_type := Word, src_type := Bool, count_type := UInt]" } GATHER_BLK(IN := #CommS2R[0], COUNT_OUT := 6, OUT => #statWordBuffer_2[0])
      { S7_Templates := "[dest_type := Bool, src_type := Word, count_type := UInt]" } SCATTER_BLK(IN := #statWordBuffer_2[0], COUNT_IN := 6, OUT => #signalsS2R.Load_Requset)
   END_RUNG
   // the same network as SCL:
   GATHER_BLK(IN := #CommS2R[0], COUNT_OUT := 6, OUT => #statWordBuffer_2[0], ENO => #_w1);
   IF #_w1 THEN
       SCATTER_BLK(IN := #statWordBuffer_2[0], COUNT_IN := 6, OUT => #signalsS2R.Load_Requset);
   END_IF;
END_REGION
END_FUNCTION_BLOCK

FUNCTION_BLOCK "GetIdentRf"   // FB96, SCL
// stored: Access Published, MemoryReserve 100, SetENOAutomatically false
   VAR_OUTPUT
      selectedRFID : USInt := 1;
      selectedAntena : USInt;
      error : Word;
   END_VAR
   VAR_IN_OUT
      identRfAllUnits : Array[*] of "typeIdentRf";   // HMI: motorstarter values
      IdentRfInterfaceHmi : "typeIdentRfHmi";
   END_VAR
   VAR
      statSelectedRfReader : USInt := 1;   // HMI: Angewählte Interface Schnittstelle (1..16) / HMI: Selected unit
      statSelectedAntena : USInt := 1;
   END_VAR
   VAR CONSTANT
      "INVALID RFID" : Word := 16#7001;   // non existant rfid
      "INVALID ANTENA" : Word := 16#7002;   // non existant antena
      OK : Word := 16#7000;
   END_VAR
BEGIN
   REGION BLOCK INFO HEADER
       //===============================================================================
       // Siemens AG / (c)Copyright 2024
       //-------------------------------------------------------------------------------
       // Title:            LAF_GetMotorstarterSignals
       // Comment/Function: This block reads diagnostic information of a Motorstarter depending
       //                   on the unit and Control Module selected in the HMI by the user.
       // Library/Family:   Automation Framework / Motorstarter Diagnostic
       // Author:           Siemens Digital Industries
       // Tested with:      S7-1517TF V3.1
       // Engineering:      TIA Portal V19
       // Restrictions:     
       //                   Required UDTs: LAF_typeDriveDiagConfig, LAF_typeDriveDiagInterfaceHmi
       // Requirements:     S7-1500(T), MC_Version V8.0
       //-------------------------------------------------------------------------------
       // Change log table:
       // Version  | Date       | Expert in charge        | Changes applied
       //----------|------------|-------------------------|-----------------------------
       // 01.00.00 | 05.06.2024 | SIMATIC Systems Support | First released version
       //===============================================================================
   END_REGION BLOCK INFO HEADER

   REGION DESCRIPTION
   (/*This block reads diagnostic information (control inputs and outputs) of a Motorstarter. 
   At runtime, this block is enabled when the ET200SP Motorstarter screen is shown in the HMI. 
   Based on the selected motorstarter object in the HMI by the user. The shown information in the HMI depends on the
   Unit and Cotrol Module selected.*/)
   END_REGION DESCRIPTION

   REGION INPUTS
       //working with static values to keep the last selected value when opening for the first time the screen  

       #statSelectedRfReader := #IdentRfInterfaceHmi.selectedRfReader;
       #statSelectedAntena := #IdentRfInterfaceHmi.selectedAntena;

   END_REGION INPUTS

   REGION ASSIGNING TEMPORARY VALUES
       // Statement section REGION
       IF #statSelectedRfReader <= "NO_OF_RF_IDENT_DEVICES" THEN
           IF #statSelectedAntena <= "NO_OF_RF_ANTENNA_DEVICES" THEN
               #IdentRfInterfaceHmi.rfReader.deviceName := #identRfAllUnits[#statSelectedRfReader].IdentRfAntena[#statSelectedAntena].deviceName;
               #IdentRfInterfaceHmi.rfReader.deviceType := #identRfAllUnits[#statSelectedRfReader].IdentRfAntena[#statSelectedAntena].deviceType;
               #IdentRfInterfaceHmi.rfReader.deviceId := #identRfAllUnits[#statSelectedRfReader].IdentRfAntena[#statSelectedAntena].deviceId;
               #IdentRfInterfaceHmi.rfReader.tagType := #identRfAllUnits[#statSelectedRfReader].IdentRfAntena[#statSelectedAntena].tagType;
               #IdentRfInterfaceHmi.rfReader.cameraMode := #identRfAllUnits[#statSelectedRfReader].IdentRfAntena[#statSelectedAntena].cameraMode;
               #IdentRfInterfaceHmi.rfReader.resultState := #identRfAllUnits[#statSelectedRfReader].IdentRfAntena[#statSelectedAntena].resultState;
               #IdentRfInterfaceHmi.rfReader.progNo := #identRfAllUnits[#statSelectedRfReader].IdentRfAntena[#statSelectedAntena].progNo;
               #IdentRfInterfaceHmi.rfReader.progNumberWrite := #identRfAllUnits[#statSelectedRfReader].IdentRfAntena[#statSelectedAntena].progNumberWrite;
               #IdentRfInterfaceHmi.rfReader.enablePushbutton := #identRfAllUnits[#statSelectedRfReader].IdentRfAntena[#statSelectedAntena].enablePushbutton;
               #IdentRfInterfaceHmi.rfReader.status := #identRfAllUnits[#statSelectedRfReader].IdentRfAntena[#statSelectedAntena].status;
               #IdentRfInterfaceHmi.rfReader.alarmCategorie := #identRfAllUnits[#statSelectedRfReader].IdentRfAntena[#statSelectedAntena].alarmCategorie;
               #IdentRfInterfaceHmi.rfReader.alarmNo := #identRfAllUnits[#statSelectedRfReader].IdentRfAntena[#statSelectedAntena].alarmNo;
               #IdentRfInterfaceHmi.rfReader.alarmCode := #identRfAllUnits[#statSelectedRfReader].IdentRfAntena[#statSelectedAntena].alarmCode;
               #IdentRfInterfaceHmi.rfReader.resultColor := #identRfAllUnits[#statSelectedRfReader].IdentRfAntena[#statSelectedAntena].resultColor;
               #IdentRfInterfaceHmi.rfReader.statusColorCode := #identRfAllUnits[#statSelectedRfReader].IdentRfAntena[#statSelectedAntena].statusColorCode;
               #IdentRfInterfaceHmi.rfReader.datRead1 := #identRfAllUnits[#statSelectedRfReader].IdentRfAntena[#statSelectedAntena].datRead1;
               #IdentRfInterfaceHmi.rfReader.datRead2 := #identRfAllUnits[#statSelectedRfReader].IdentRfAntena[#statSelectedAntena].datRead2;
               #IdentRfInterfaceHmi.rfReader.datRead3 := #identRfAllUnits[#statSelectedRfReader].IdentRfAntena[#statSelectedAntena].datRead3;
               #IdentRfInterfaceHmi.rfReader.datRead4 := #identRfAllUnits[#statSelectedRfReader].IdentRfAntena[#statSelectedAntena].datRead4;

               #identRfAllUnits[#statSelectedRfReader].IdentRfAntena[#statSelectedAntena].pushbutton := #IdentRfInterfaceHmi.rfReader.pushbutton;
               #identRfAllUnits[#statSelectedRfReader].IdentRfAntena[#statSelectedAntena].datWrite1 := #IdentRfInterfaceHmi.rfReader.datWrite1;
               #identRfAllUnits[#statSelectedRfReader].IdentRfAntena[#statSelectedAntena].datWrite2 := #IdentRfInterfaceHmi.rfReader.datWrite2;
               #identRfAllUnits[#statSelectedRfReader].IdentRfAntena[#statSelectedAntena].datWrite3 := #IdentRfInterfaceHmi.rfReader.datWrite3;
               #identRfAllUnits[#statSelectedRfReader].IdentRfAntena[#statSelectedAntena].datWrite4 := #IdentRfInterfaceHmi.rfReader.datWrite4;

               #error := #OK;
           ELSE
               #error := #"INVALID ANTENA";
           END_IF;

       ELSE
           #error := #"INVALID RFID";
       END_IF;

   END_REGION


   REGION OUTPUTS
       // Statement section REGION
       #selectedAntena := #statSelectedAntena;
       #selectedRFID := #statSelectedRfReader;
   END_REGION
END_FUNCTION_BLOCK

FUNCTION "Safety Door" : Void   // FC97, LAD
// stored: SetENOAutomatically false
   VAR CONSTANT
      TRUE : Bool := TRUE;
      FALSE : Bool;
   END_VAR
   VAR_TEMP   // added for the SCL form of the ladder/FBD networks
      _w1 : Bool;
   END_VAR
BEGIN

REGION Network 1: FDoorEC.TOP Monitoring
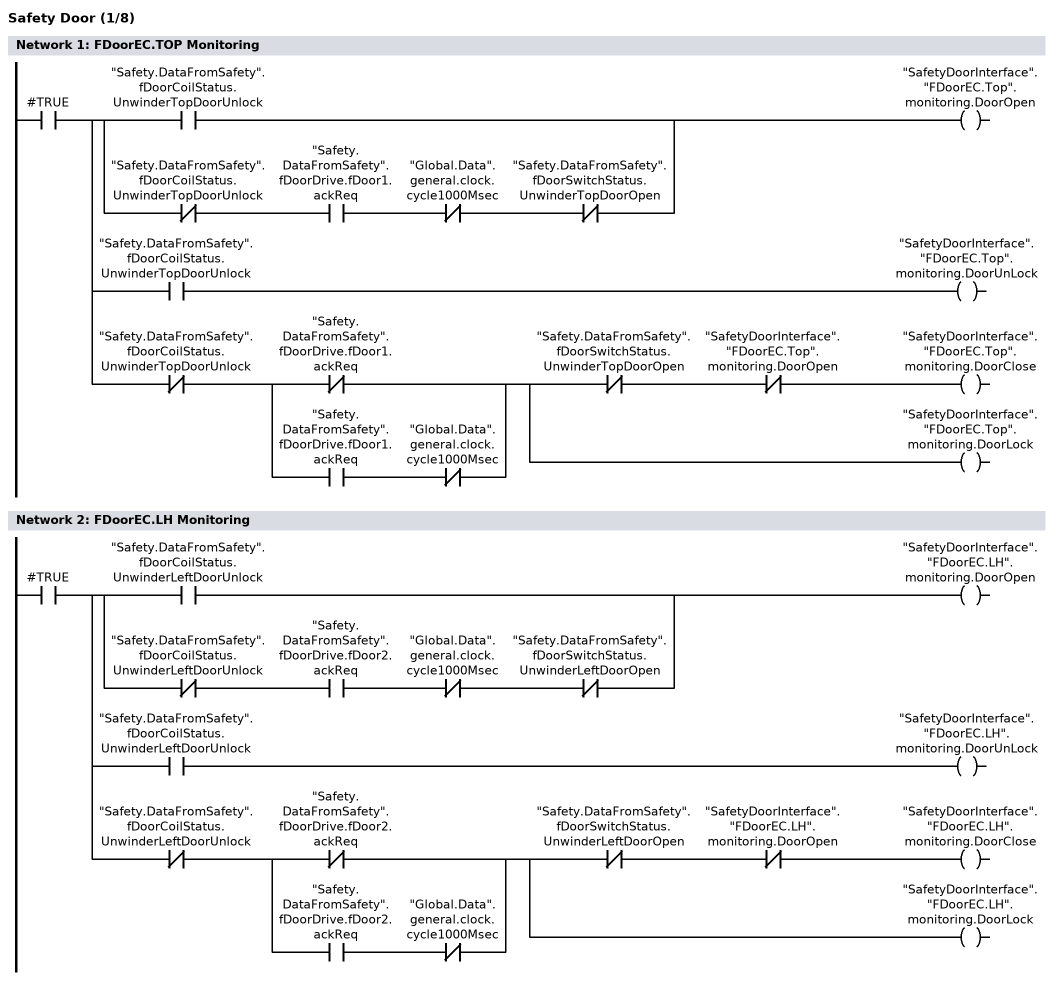
   RUNG wire#powerrail
      Contact( #TRUE )
      wire#w1
      Contact( "Safety.DataFromSafety".fDoorCoilStatus.UnwinderTopDoorUnlock )
      wire#w2
      Coil( "SafetyDoorInterface"."FDoorEC.Top".monitoring.DoorOpen )
   END_RUNG
   RUNG wire#w1
      I_Contact( "Safety.DataFromSafety".fDoorCoilStatus.UnwinderTopDoorUnlock )
      Contact( "Safety.DataFromSafety".fDoorDrive.fDoor1.ackReq )
      I_Contact( "Global.Data".general.clock.cycle1000Msec )
      I_Contact( "Safety.DataFromSafety".fDoorSwitchStatus.UnwinderTopDoorOpen )
   END_RUNG wire#w2
   RUNG wire#w1
      Contact( "Safety.DataFromSafety".fDoorCoilStatus.UnwinderTopDoorUnlock )
      Coil( "SafetyDoorInterface"."FDoorEC.Top".monitoring.DoorUnLock )
   END_RUNG
   RUNG wire#w1
      I_Contact( "Safety.DataFromSafety".fDoorCoilStatus.UnwinderTopDoorUnlock )
      wire#w3
      I_Contact( "Safety.DataFromSafety".fDoorDrive.fDoor1.ackReq )
      wire#w4
      I_Contact( "Safety.DataFromSafety".fDoorSwitchStatus.UnwinderTopDoorOpen )
      I_Contact( "SafetyDoorInterface"."FDoorEC.Top".monitoring.DoorOpen )
      Coil( "SafetyDoorInterface"."FDoorEC.Top".monitoring.DoorClose )
   END_RUNG
   RUNG wire#w3
      Contact( "Safety.DataFromSafety".fDoorDrive.fDoor1.ackReq )
      I_Contact( "Global.Data".general.clock.cycle1000Msec )
   END_RUNG wire#w4
   RUNG wire#w4
      Coil( "SafetyDoorInterface"."FDoorEC.Top".monitoring.DoorLock )
   END_RUNG
   // the same network as SCL:
   "SafetyDoorInterface"."FDoorEC.Top".monitoring.DoorOpen := #TRUE AND ("Safety.DataFromSafety".fDoorCoilStatus.UnwinderTopDoorUnlock OR (NOT "Safety.DataFromSafety".fDoorCoilStatus.UnwinderTopDoorUnlock AND "Safety.DataFromSafety".fDoorDrive.fDoor1.ackReq AND NOT "Global.Data".general.clock.cycle1000Msec AND NOT "Safety.DataFromSafety".fDoorSwitchStatus.UnwinderTopDoorOpen));
   "SafetyDoorInterface"."FDoorEC.Top".monitoring.DoorUnLock := #TRUE AND "Safety.DataFromSafety".fDoorCoilStatus.UnwinderTopDoorUnlock;
   #_w1 := #TRUE AND NOT "Safety.DataFromSafety".fDoorCoilStatus.UnwinderTopDoorUnlock AND (NOT "Safety.DataFromSafety".fDoorDrive.fDoor1.ackReq OR ("Safety.DataFromSafety".fDoorDrive.fDoor1.ackReq AND NOT "Global.Data".general.clock.cycle1000Msec));
   "SafetyDoorInterface"."FDoorEC.Top".monitoring.DoorClose := #_w1 AND NOT "Safety.DataFromSafety".fDoorSwitchStatus.UnwinderTopDoorOpen AND NOT "SafetyDoorInterface"."FDoorEC.Top".monitoring.DoorOpen;
   "SafetyDoorInterface"."FDoorEC.Top".monitoring.DoorLock := #_w1;
END_REGION

REGION Network 2: FDoorEC.LH Monitoring
   RUNG wire#powerrail
      Contact( #TRUE )
      wire#w1
      Contact( "Safety.DataFromSafety".fDoorCoilStatus.UnwinderLeftDoorUnlock )
      wire#w2
      Coil( "SafetyDoorInterface"."FDoorEC.LH".monitoring.DoorOpen )
   END_RUNG
   RUNG wire#w1
      I_Contact( "Safety.DataFromSafety".fDoorCoilStatus.UnwinderLeftDoorUnlock )
      Contact( "Safety.DataFromSafety".fDoorDrive.fDoor2.ackReq )
      I_Contact( "Global.Data".general.clock.cycle1000Msec )
      I_Contact( "Safety.DataFromSafety".fDoorSwitchStatus.UnwinderLeftDoorOpen )
   END_RUNG wire#w2
   RUNG wire#w1
      Contact( "Safety.DataFromSafety".fDoorCoilStatus.UnwinderLeftDoorUnlock )
      Coil( "SafetyDoorInterface"."FDoorEC.LH".monitoring.DoorUnLock )
   END_RUNG
   RUNG wire#w1
      I_Contact( "Safety.DataFromSafety".fDoorCoilStatus.UnwinderLeftDoorUnlock )
      wire#w3
      I_Contact( "Safety.DataFromSafety".fDoorDrive.fDoor2.ackReq )
      wire#w4
      I_Contact( "Safety.DataFromSafety".fDoorSwitchStatus.UnwinderLeftDoorOpen )
      I_Contact( "SafetyDoorInterface"."FDoorEC.LH".monitoring.DoorOpen )
      Coil( "SafetyDoorInterface"."FDoorEC.LH".monitoring.DoorClose )
   END_RUNG
   RUNG wire#w3
      Contact( "Safety.DataFromSafety".fDoorDrive.fDoor2.ackReq )
      I_Contact( "Global.Data".general.clock.cycle1000Msec )
   END_RUNG wire#w4
   RUNG wire#w4
      Coil( "SafetyDoorInterface"."FDoorEC.LH".monitoring.DoorLock )
   END_RUNG
   // the same network as SCL:
   "SafetyDoorInterface"."FDoorEC.LH".monitoring.DoorOpen := #TRUE AND ("Safety.DataFromSafety".fDoorCoilStatus.UnwinderLeftDoorUnlock OR (NOT "Safety.DataFromSafety".fDoorCoilStatus.UnwinderLeftDoorUnlock AND "Safety.DataFromSafety".fDoorDrive.fDoor2.ackReq AND NOT "Global.Data".general.clock.cycle1000Msec AND NOT "Safety.DataFromSafety".fDoorSwitchStatus.UnwinderLeftDoorOpen));
   "SafetyDoorInterface"."FDoorEC.LH".monitoring.DoorUnLock := #TRUE AND "Safety.DataFromSafety".fDoorCoilStatus.UnwinderLeftDoorUnlock;
   #_w1 := #TRUE AND NOT "Safety.DataFromSafety".fDoorCoilStatus.UnwinderLeftDoorUnlock AND (NOT "Safety.DataFromSafety".fDoorDrive.fDoor2.ackReq OR ("Safety.DataFromSafety".fDoorDrive.fDoor2.ackReq AND NOT "Global.Data".general.clock.cycle1000Msec));
   "SafetyDoorInterface"."FDoorEC.LH".monitoring.DoorClose := #_w1 AND NOT "Safety.DataFromSafety".fDoorSwitchStatus.UnwinderLeftDoorOpen AND NOT "SafetyDoorInterface"."FDoorEC.LH".monitoring.DoorOpen;
   "SafetyDoorInterface"."FDoorEC.LH".monitoring.DoorLock := #_w1;
END_REGION

REGION Network 3: FDoorEC.RH Monitoring
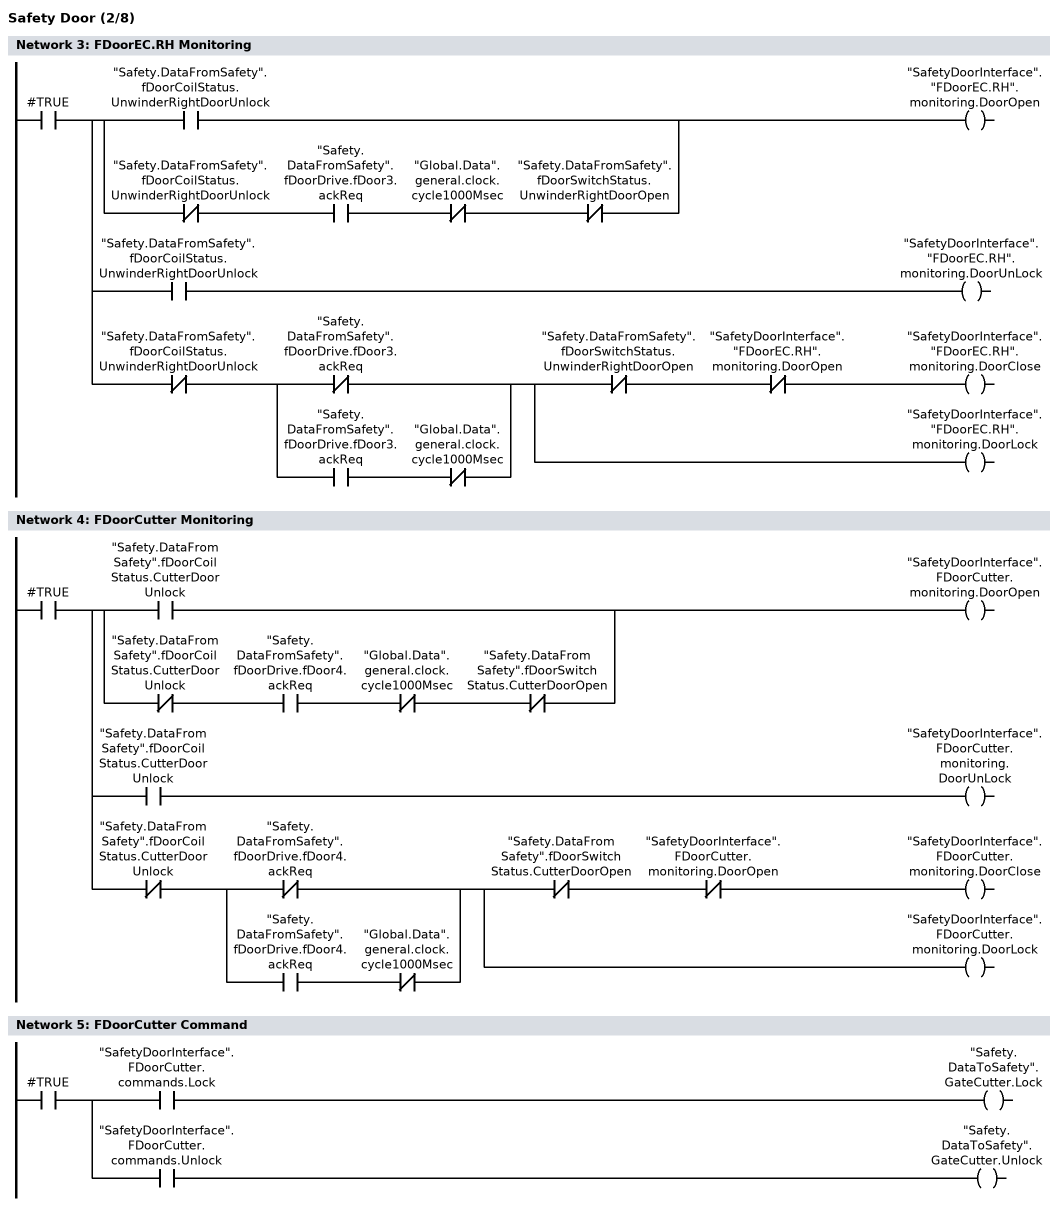
   RUNG wire#powerrail
      Contact( #TRUE )
      wire#w1
      Contact( "Safety.DataFromSafety".fDoorCoilStatus.UnwinderRightDoorUnlock )
      wire#w2
      Coil( "SafetyDoorInterface"."FDoorEC.RH".monitoring.DoorOpen )
   END_RUNG
   RUNG wire#w1
      I_Contact( "Safety.DataFromSafety".fDoorCoilStatus.UnwinderRightDoorUnlock )
      Contact( "Safety.DataFromSafety".fDoorDrive.fDoor3.ackReq )
      I_Contact( "Global.Data".general.clock.cycle1000Msec )
      I_Contact( "Safety.DataFromSafety".fDoorSwitchStatus.UnwinderRightDoorOpen )
   END_RUNG wire#w2
   RUNG wire#w1
      Contact( "Safety.DataFromSafety".fDoorCoilStatus.UnwinderRightDoorUnlock )
      Coil( "SafetyDoorInterface"."FDoorEC.RH".monitoring.DoorUnLock )
   END_RUNG
   RUNG wire#w1
      I_Contact( "Safety.DataFromSafety".fDoorCoilStatus.UnwinderRightDoorUnlock )
      wire#w3
      I_Contact( "Safety.DataFromSafety".fDoorDrive.fDoor3.ackReq )
      wire#w4
      I_Contact( "Safety.DataFromSafety".fDoorSwitchStatus.UnwinderRightDoorOpen )
      I_Contact( "SafetyDoorInterface"."FDoorEC.RH".monitoring.DoorOpen )
      Coil( "SafetyDoorInterface"."FDoorEC.RH".monitoring.DoorClose )
   END_RUNG
   RUNG wire#w3
      Contact( "Safety.DataFromSafety".fDoorDrive.fDoor3.ackReq )
      I_Contact( "Global.Data".general.clock.cycle1000Msec )
   END_RUNG wire#w4
   RUNG wire#w4
      Coil( "SafetyDoorInterface"."FDoorEC.RH".monitoring.DoorLock )
   END_RUNG
   // the same network as SCL:
   "SafetyDoorInterface"."FDoorEC.RH".monitoring.DoorOpen := #TRUE AND ("Safety.DataFromSafety".fDoorCoilStatus.UnwinderRightDoorUnlock OR (NOT "Safety.DataFromSafety".fDoorCoilStatus.UnwinderRightDoorUnlock AND "Safety.DataFromSafety".fDoorDrive.fDoor3.ackReq AND NOT "Global.Data".general.clock.cycle1000Msec AND NOT "Safety.DataFromSafety".fDoorSwitchStatus.UnwinderRightDoorOpen));
   "SafetyDoorInterface"."FDoorEC.RH".monitoring.DoorUnLock := #TRUE AND "Safety.DataFromSafety".fDoorCoilStatus.UnwinderRightDoorUnlock;
   #_w1 := #TRUE AND NOT "Safety.DataFromSafety".fDoorCoilStatus.UnwinderRightDoorUnlock AND (NOT "Safety.DataFromSafety".fDoorDrive.fDoor3.ackReq OR ("Safety.DataFromSafety".fDoorDrive.fDoor3.ackReq AND NOT "Global.Data".general.clock.cycle1000Msec));
   "SafetyDoorInterface"."FDoorEC.RH".monitoring.DoorClose := #_w1 AND NOT "Safety.DataFromSafety".fDoorSwitchStatus.UnwinderRightDoorOpen AND NOT "SafetyDoorInterface"."FDoorEC.RH".monitoring.DoorOpen;
   "SafetyDoorInterface"."FDoorEC.RH".monitoring.DoorLock := #_w1;
END_REGION

REGION Network 4: FDoorCutter Monitoring
   RUNG wire#powerrail
      Contact( #TRUE )
      wire#w1
      Contact( "Safety.DataFromSafety".fDoorCoilStatus.CutterDoorUnlock )
      wire#w2
      Coil( "SafetyDoorInterface".FDoorCutter.monitoring.DoorOpen )
   END_RUNG
   RUNG wire#w1
      I_Contact( "Safety.DataFromSafety".fDoorCoilStatus.CutterDoorUnlock )
      Contact( "Safety.DataFromSafety".fDoorDrive.fDoor4.ackReq )
      I_Contact( "Global.Data".general.clock.cycle1000Msec )
      I_Contact( "Safety.DataFromSafety".fDoorSwitchStatus.CutterDoorOpen )
   END_RUNG wire#w2
   RUNG wire#w1
      Contact( "Safety.DataFromSafety".fDoorCoilStatus.CutterDoorUnlock )
      Coil( "SafetyDoorInterface".FDoorCutter.monitoring.DoorUnLock )
   END_RUNG
   RUNG wire#w1
      I_Contact( "Safety.DataFromSafety".fDoorCoilStatus.CutterDoorUnlock )
      wire#w3
      I_Contact( "Safety.DataFromSafety".fDoorDrive.fDoor4.ackReq )
      wire#w4
      I_Contact( "Safety.DataFromSafety".fDoorSwitchStatus.CutterDoorOpen )
      I_Contact( "SafetyDoorInterface".FDoorCutter.monitoring.DoorOpen )
      Coil( "SafetyDoorInterface".FDoorCutter.monitoring.DoorClose )
   END_RUNG
   RUNG wire#w3
      Contact( "Safety.DataFromSafety".fDoorDrive.fDoor4.ackReq )
      I_Contact( "Global.Data".general.clock.cycle1000Msec )
   END_RUNG wire#w4
   RUNG wire#w4
      Coil( "SafetyDoorInterface".FDoorCutter.monitoring.DoorLock )
   END_RUNG
   // the same network as SCL:
   "SafetyDoorInterface".FDoorCutter.monitoring.DoorOpen := #TRUE AND ("Safety.DataFromSafety".fDoorCoilStatus.CutterDoorUnlock OR (NOT "Safety.DataFromSafety".fDoorCoilStatus.CutterDoorUnlock AND "Safety.DataFromSafety".fDoorDrive.fDoor4.ackReq AND NOT "Global.Data".general.clock.cycle1000Msec AND NOT "Safety.DataFromSafety".fDoorSwitchStatus.CutterDoorOpen));
   "SafetyDoorInterface".FDoorCutter.monitoring.DoorUnLock := #TRUE AND "Safety.DataFromSafety".fDoorCoilStatus.CutterDoorUnlock;
   #_w1 := #TRUE AND NOT "Safety.DataFromSafety".fDoorCoilStatus.CutterDoorUnlock AND (NOT "Safety.DataFromSafety".fDoorDrive.fDoor4.ackReq OR ("Safety.DataFromSafety".fDoorDrive.fDoor4.ackReq AND NOT "Global.Data".general.clock.cycle1000Msec));
   "SafetyDoorInterface".FDoorCutter.monitoring.DoorClose := #_w1 AND NOT "Safety.DataFromSafety".fDoorSwitchStatus.CutterDoorOpen AND NOT "SafetyDoorInterface".FDoorCutter.monitoring.DoorOpen;
   "SafetyDoorInterface".FDoorCutter.monitoring.DoorLock := #_w1;
END_REGION

REGION Network 5: FDoorCutter Command
   RUNG wire#powerrail
      Contact( #TRUE )
      wire#w1
      Contact( "SafetyDoorInterface".FDoorCutter.commands.Lock )
      Coil( "Safety.DataToSafety".GateCutter.Lock )
   END_RUNG
   RUNG wire#w1
      Contact( "SafetyDoorInterface".FDoorCutter.commands.Unlock )
      Coil( "Safety.DataToSafety".GateCutter.Unlock )
   END_RUNG
   // the same network as SCL:
   "Safety.DataToSafety".GateCutter.Lock := #TRUE AND "SafetyDoorInterface".FDoorCutter.commands.Lock;
   "Safety.DataToSafety".GateCutter.Unlock := #TRUE AND "SafetyDoorInterface".FDoorCutter.commands.Unlock;
END_REGION

REGION Network 6: FDoorMagazine Monitoring
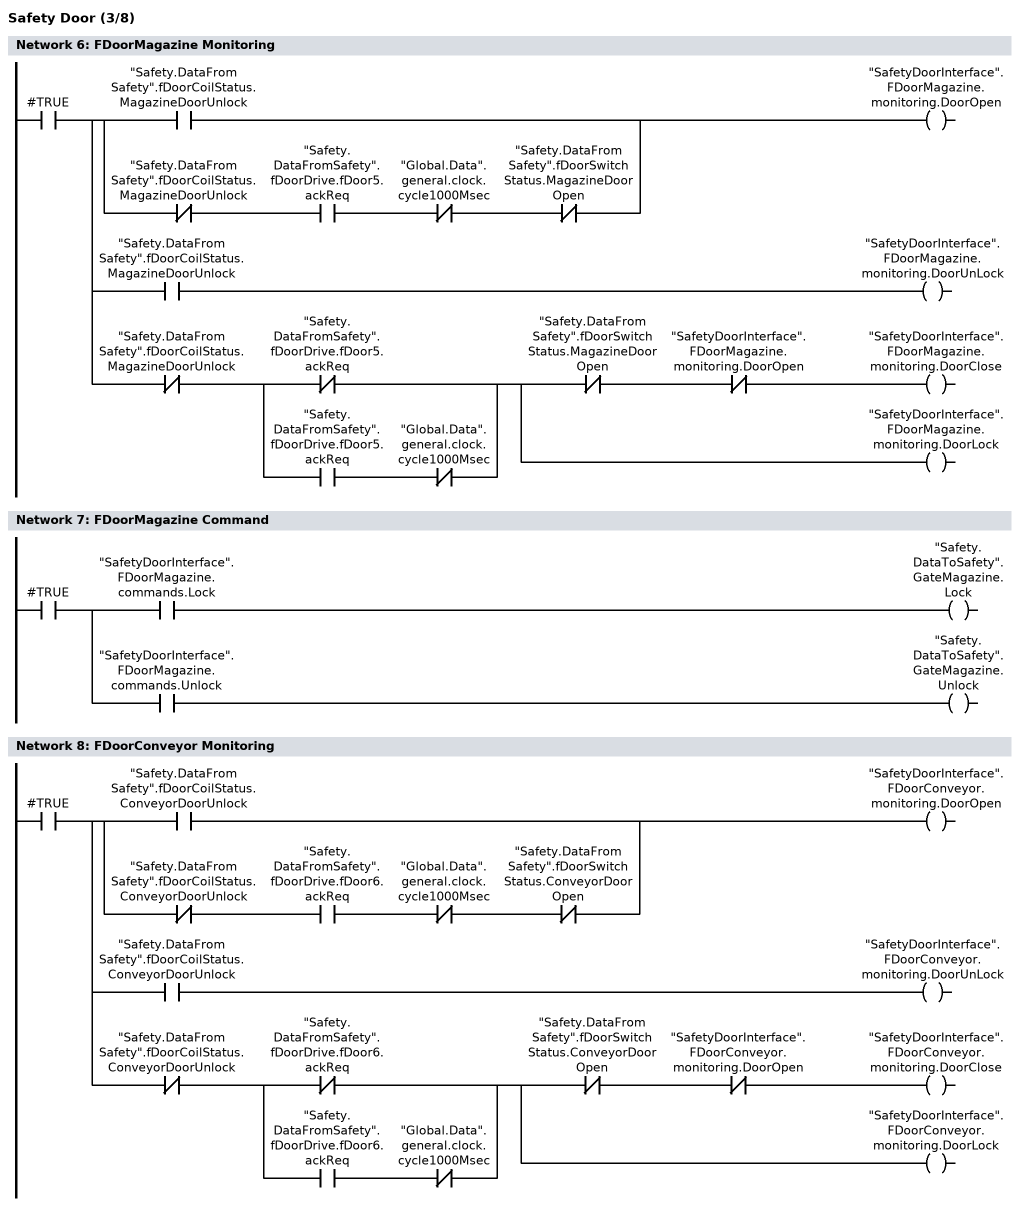
   RUNG wire#powerrail
      Contact( #TRUE )
      wire#w1
      Contact( "Safety.DataFromSafety".fDoorCoilStatus.MagazineDoorUnlock )
      wire#w2
      Coil( "SafetyDoorInterface".FDoorMagazine.monitoring.DoorOpen )
   END_RUNG
   RUNG wire#w1
      I_Contact( "Safety.DataFromSafety".fDoorCoilStatus.MagazineDoorUnlock )
      Contact( "Safety.DataFromSafety".fDoorDrive.fDoor5.ackReq )
      I_Contact( "Global.Data".general.clock.cycle1000Msec )
      I_Contact( "Safety.DataFromSafety".fDoorSwitchStatus.MagazineDoorOpen )
   END_RUNG wire#w2
   RUNG wire#w1
      Contact( "Safety.DataFromSafety".fDoorCoilStatus.MagazineDoorUnlock )
      Coil( "SafetyDoorInterface".FDoorMagazine.monitoring.DoorUnLock )
   END_RUNG
   RUNG wire#w1
      I_Contact( "Safety.DataFromSafety".fDoorCoilStatus.MagazineDoorUnlock )
      wire#w3
      I_Contact( "Safety.DataFromSafety".fDoorDrive.fDoor5.ackReq )
      wire#w4
      I_Contact( "Safety.DataFromSafety".fDoorSwitchStatus.MagazineDoorOpen )
      I_Contact( "SafetyDoorInterface".FDoorMagazine.monitoring.DoorOpen )
      Coil( "SafetyDoorInterface".FDoorMagazine.monitoring.DoorClose )
   END_RUNG
   RUNG wire#w3
      Contact( "Safety.DataFromSafety".fDoorDrive.fDoor5.ackReq )
      I_Contact( "Global.Data".general.clock.cycle1000Msec )
   END_RUNG wire#w4
   RUNG wire#w4
      Coil( "SafetyDoorInterface".FDoorMagazine.monitoring.DoorLock )
   END_RUNG
   // the same network as SCL:
   "SafetyDoorInterface".FDoorMagazine.monitoring.DoorOpen := #TRUE AND ("Safety.DataFromSafety".fDoorCoilStatus.MagazineDoorUnlock OR (NOT "Safety.DataFromSafety".fDoorCoilStatus.MagazineDoorUnlock AND "Safety.DataFromSafety".fDoorDrive.fDoor5.ackReq AND NOT "Global.Data".general.clock.cycle1000Msec AND NOT "Safety.DataFromSafety".fDoorSwitchStatus.MagazineDoorOpen));
   "SafetyDoorInterface".FDoorMagazine.monitoring.DoorUnLock := #TRUE AND "Safety.DataFromSafety".fDoorCoilStatus.MagazineDoorUnlock;
   #_w1 := #TRUE AND NOT "Safety.DataFromSafety".fDoorCoilStatus.MagazineDoorUnlock AND (NOT "Safety.DataFromSafety".fDoorDrive.fDoor5.ackReq OR ("Safety.DataFromSafety".fDoorDrive.fDoor5.ackReq AND NOT "Global.Data".general.clock.cycle1000Msec));
   "SafetyDoorInterface".FDoorMagazine.monitoring.DoorClose := #_w1 AND NOT "Safety.DataFromSafety".fDoorSwitchStatus.MagazineDoorOpen AND NOT "SafetyDoorInterface".FDoorMagazine.monitoring.DoorOpen;
   "SafetyDoorInterface".FDoorMagazine.monitoring.DoorLock := #_w1;
END_REGION

REGION Network 7: FDoorMagazine Command
   RUNG wire#powerrail
      Contact( #TRUE )
      wire#w1
      Contact( "SafetyDoorInterface".FDoorMagazine.commands.Lock )
      Coil( "Safety.DataToSafety".GateMagazine.Lock )
   END_RUNG
   RUNG wire#w1
      Contact( "SafetyDoorInterface".FDoorMagazine.commands.Unlock )
      Coil( "Safety.DataToSafety".GateMagazine.Unlock )
   END_RUNG
   // the same network as SCL:
   "Safety.DataToSafety".GateMagazine.Lock := #TRUE AND "SafetyDoorInterface".FDoorMagazine.commands.Lock;
   "Safety.DataToSafety".GateMagazine.Unlock := #TRUE AND "SafetyDoorInterface".FDoorMagazine.commands.Unlock;
END_REGION

REGION Network 8: FDoorConveyor Monitoring
   RUNG wire#powerrail
      Contact( #TRUE )
      wire#w1
      Contact( "Safety.DataFromSafety".fDoorCoilStatus.ConveyorDoorUnlock )
      wire#w2
      Coil( "SafetyDoorInterface".FDoorConveyor.monitoring.DoorOpen )
   END_RUNG
   RUNG wire#w1
      I_Contact( "Safety.DataFromSafety".fDoorCoilStatus.ConveyorDoorUnlock )
      Contact( "Safety.DataFromSafety".fDoorDrive.fDoor6.ackReq )
      I_Contact( "Global.Data".general.clock.cycle1000Msec )
      I_Contact( "Safety.DataFromSafety".fDoorSwitchStatus.ConveyorDoorOpen )
   END_RUNG wire#w2
   RUNG wire#w1
      Contact( "Safety.DataFromSafety".fDoorCoilStatus.ConveyorDoorUnlock )
      Coil( "SafetyDoorInterface".FDoorConveyor.monitoring.DoorUnLock )
   END_RUNG
   RUNG wire#w1
      I_Contact( "Safety.DataFromSafety".fDoorCoilStatus.ConveyorDoorUnlock )
      wire#w3
      I_Contact( "Safety.DataFromSafety".fDoorDrive.fDoor6.ackReq )
      wire#w4
      I_Contact( "Safety.DataFromSafety".fDoorSwitchStatus.ConveyorDoorOpen )
      I_Contact( "SafetyDoorInterface".FDoorConveyor.monitoring.DoorOpen )
      Coil( "SafetyDoorInterface".FDoorConveyor.monitoring.DoorClose )
   END_RUNG
   RUNG wire#w3
      Contact( "Safety.DataFromSafety".fDoorDrive.fDoor6.ackReq )
      I_Contact( "Global.Data".general.clock.cycle1000Msec )
   END_RUNG wire#w4
   RUNG wire#w4
      Coil( "SafetyDoorInterface".FDoorConveyor.monitoring.DoorLock )
   END_RUNG
   // the same network as SCL:
   "SafetyDoorInterface".FDoorConveyor.monitoring.DoorOpen := #TRUE AND ("Safety.DataFromSafety".fDoorCoilStatus.ConveyorDoorUnlock OR (NOT "Safety.DataFromSafety".fDoorCoilStatus.ConveyorDoorUnlock AND "Safety.DataFromSafety".fDoorDrive.fDoor6.ackReq AND NOT "Global.Data".general.clock.cycle1000Msec AND NOT "Safety.DataFromSafety".fDoorSwitchStatus.ConveyorDoorOpen));
   "SafetyDoorInterface".FDoorConveyor.monitoring.DoorUnLock := #TRUE AND "Safety.DataFromSafety".fDoorCoilStatus.ConveyorDoorUnlock;
   #_w1 := #TRUE AND NOT "Safety.DataFromSafety".fDoorCoilStatus.ConveyorDoorUnlock AND (NOT "Safety.DataFromSafety".fDoorDrive.fDoor6.ackReq OR ("Safety.DataFromSafety".fDoorDrive.fDoor6.ackReq AND NOT "Global.Data".general.clock.cycle1000Msec));
   "SafetyDoorInterface".FDoorConveyor.monitoring.DoorClose := #_w1 AND NOT "Safety.DataFromSafety".fDoorSwitchStatus.ConveyorDoorOpen AND NOT "SafetyDoorInterface".FDoorConveyor.monitoring.DoorOpen;
   "SafetyDoorInterface".FDoorConveyor.monitoring.DoorLock := #_w1;
END_REGION

REGION Network 9: FDoorConveyor Command
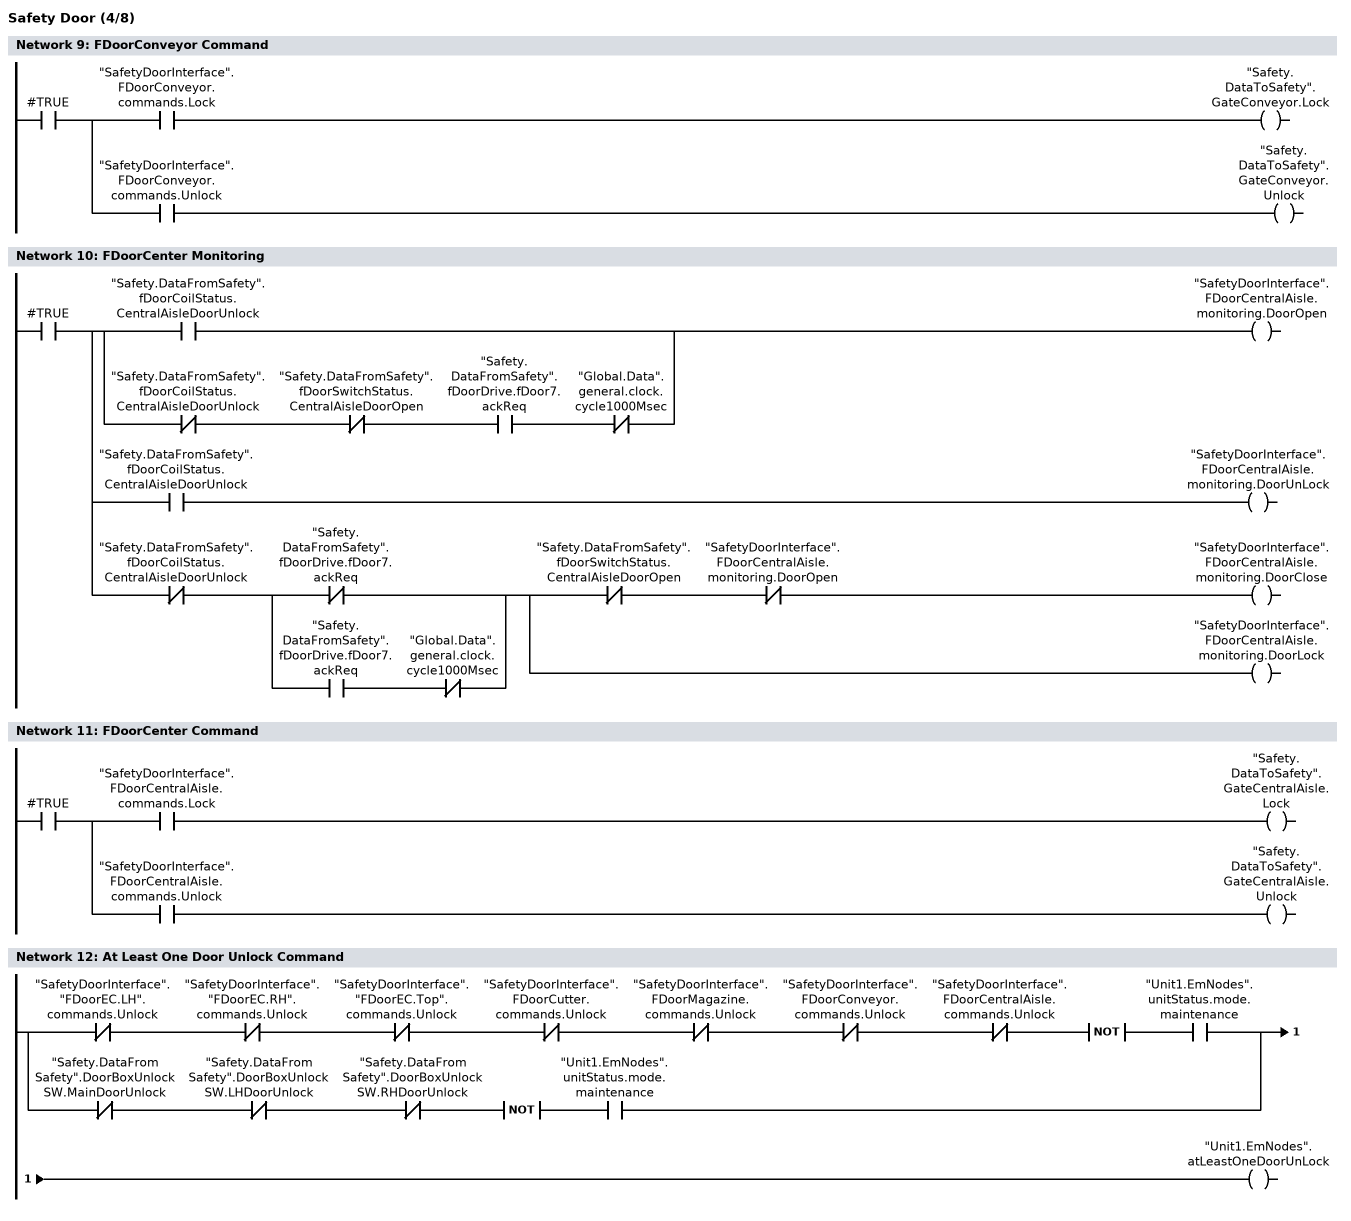
   RUNG wire#powerrail
      Contact( #TRUE )
      wire#w1
      Contact( "SafetyDoorInterface".FDoorConveyor.commands.Lock )
      Coil( "Safety.DataToSafety".GateConveyor.Lock )
   END_RUNG
   RUNG wire#w1
      Contact( "SafetyDoorInterface".FDoorConveyor.commands.Unlock )
      Coil( "Safety.DataToSafety".GateConveyor.Unlock )
   END_RUNG
   // the same network as SCL:
   "Safety.DataToSafety".GateConveyor.Lock := #TRUE AND "SafetyDoorInterface".FDoorConveyor.commands.Lock;
   "Safety.DataToSafety".GateConveyor.Unlock := #TRUE AND "SafetyDoorInterface".FDoorConveyor.commands.Unlock;
END_REGION

REGION Network 10: FDoorCenter Monitoring
   RUNG wire#powerrail
      Contact( #TRUE )
      wire#w1
      Contact( "Safety.DataFromSafety".fDoorCoilStatus.CentralAisleDoorUnlock )
      wire#w2
      Coil( "SafetyDoorInterface".FDoorCentralAisle.monitoring.DoorOpen )
   END_RUNG
   RUNG wire#w1
      I_Contact( "Safety.DataFromSafety".fDoorCoilStatus.CentralAisleDoorUnlock )
      I_Contact( "Safety.DataFromSafety".fDoorSwitchStatus.CentralAisleDoorOpen )
      Contact( "Safety.DataFromSafety".fDoorDrive.fDoor7.ackReq )
      I_Contact( "Global.Data".general.clock.cycle1000Msec )
   END_RUNG wire#w2
   RUNG wire#w1
      Contact( "Safety.DataFromSafety".fDoorCoilStatus.CentralAisleDoorUnlock )
      Coil( "SafetyDoorInterface".FDoorCentralAisle.monitoring.DoorUnLock )
   END_RUNG
   RUNG wire#w1
      I_Contact( "Safety.DataFromSafety".fDoorCoilStatus.CentralAisleDoorUnlock )
      wire#w3
      I_Contact( "Safety.DataFromSafety".fDoorDrive.fDoor7.ackReq )
      wire#w4
      I_Contact( "Safety.DataFromSafety".fDoorSwitchStatus.CentralAisleDoorOpen )
      I_Contact( "SafetyDoorInterface".FDoorCentralAisle.monitoring.DoorOpen )
      Coil( "SafetyDoorInterface".FDoorCentralAisle.monitoring.DoorClose )
   END_RUNG
   RUNG wire#w3
      Contact( "Safety.DataFromSafety".fDoorDrive.fDoor7.ackReq )
      I_Contact( "Global.Data".general.clock.cycle1000Msec )
   END_RUNG wire#w4
   RUNG wire#w4
      Coil( "SafetyDoorInterface".FDoorCentralAisle.monitoring.DoorLock )
   END_RUNG
   // the same network as SCL:
   "SafetyDoorInterface".FDoorCentralAisle.monitoring.DoorOpen := #TRUE AND ("Safety.DataFromSafety".fDoorCoilStatus.CentralAisleDoorUnlock OR (NOT "Safety.DataFromSafety".fDoorCoilStatus.CentralAisleDoorUnlock AND NOT "Safety.DataFromSafety".fDoorSwitchStatus.CentralAisleDoorOpen AND "Safety.DataFromSafety".fDoorDrive.fDoor7.ackReq AND NOT "Global.Data".general.clock.cycle1000Msec));
   "SafetyDoorInterface".FDoorCentralAisle.monitoring.DoorUnLock := #TRUE AND "Safety.DataFromSafety".fDoorCoilStatus.CentralAisleDoorUnlock;
   #_w1 := #TRUE AND NOT "Safety.DataFromSafety".fDoorCoilStatus.CentralAisleDoorUnlock AND (NOT "Safety.DataFromSafety".fDoorDrive.fDoor7.ackReq OR ("Safety.DataFromSafety".fDoorDrive.fDoor7.ackReq AND NOT "Global.Data".general.clock.cycle1000Msec));
   "SafetyDoorInterface".FDoorCentralAisle.monitoring.DoorClose := #_w1 AND NOT "Safety.DataFromSafety".fDoorSwitchStatus.CentralAisleDoorOpen AND NOT "SafetyDoorInterface".FDoorCentralAisle.monitoring.DoorOpen;
   "SafetyDoorInterface".FDoorCentralAisle.monitoring.DoorLock := #_w1;
END_REGION

REGION Network 11: FDoorCenter Command
   RUNG wire#powerrail
      Contact( #TRUE )
      wire#w1
      Contact( "SafetyDoorInterface".FDoorCentralAisle.commands.Lock )
      Coil( "Safety.DataToSafety".GateCentralAisle.Lock )
   END_RUNG
   RUNG wire#w1
      Contact( "SafetyDoorInterface".FDoorCentralAisle.commands.Unlock )
      Coil( "Safety.DataToSafety".GateCentralAisle.Unlock )
   END_RUNG
   // the same network as SCL:
   "Safety.DataToSafety".GateCentralAisle.Lock := #TRUE AND "SafetyDoorInterface".FDoorCentralAisle.commands.Lock;
   "Safety.DataToSafety".GateCentralAisle.Unlock := #TRUE AND "SafetyDoorInterface".FDoorCentralAisle.commands.Unlock;
END_REGION

REGION Network 12: At Least One Door Unlock Command
   RUNG wire#powerrail
      I_Contact( "SafetyDoorInterface"."FDoorEC.LH".commands.Unlock )
      I_Contact( "SafetyDoorInterface"."FDoorEC.RH".commands.Unlock )
      I_Contact( "SafetyDoorInterface"."FDoorEC.Top".commands.Unlock )
      I_Contact( "SafetyDoorInterface".FDoorCutter.commands.Unlock )
      I_Contact( "SafetyDoorInterface".FDoorMagazine.commands.Unlock )
      I_Contact( "SafetyDoorInterface".FDoorConveyor.commands.Unlock )
      I_Contact( "SafetyDoorInterface".FDoorCentralAisle.commands.Unlock )
      Not()
      Contact( "Unit1.EmNodes".unitStatus.mode.maintenance )
      wire#w1
      Coil( "Unit1.EmNodes".atLeastOneDoorUnLock )
   END_RUNG
   RUNG wire#powerrail
      I_Contact( "Safety.DataFromSafety".DoorBoxUnlockSW.MainDoorUnlock )
      I_Contact( "Safety.DataFromSafety".DoorBoxUnlockSW.LHDoorUnlock )
      I_Contact( "Safety.DataFromSafety".DoorBoxUnlockSW.RHDoorUnlock )
      Not()
      Contact( "Unit1.EmNodes".unitStatus.mode.maintenance )
   END_RUNG wire#w1
   // the same network as SCL:
   "Unit1.EmNodes".atLeastOneDoorUnLock := (NOT (NOT "SafetyDoorInterface"."FDoorEC.LH".commands.Unlock AND NOT "SafetyDoorInterface"."FDoorEC.RH".commands.Unlock AND NOT "SafetyDoorInterface"."FDoorEC.Top".commands.Unlock AND NOT "SafetyDoorInterface".FDoorCutter.commands.Unlock AND NOT "SafetyDoorInterface".FDoorMagazine.commands.Unlock AND NOT "SafetyDoorInterface".FDoorConveyor.commands.Unlock AND NOT "SafetyDoorInterface".FDoorCentralAisle.commands.Unlock) AND "Unit1.EmNodes".unitStatus.mode.maintenance) OR (NOT (NOT "Safety.DataFromSafety".DoorBoxUnlockSW.MainDoorUnlock AND NOT "Safety.DataFromSafety".DoorBoxUnlockSW.LHDoorUnlock AND NOT "Safety.DataFromSafety".DoorBoxUnlockSW.RHDoorUnlock) AND "Unit1.EmNodes".unitStatus.mode.maintenance);
END_REGION

REGION Network 13: OtherDoor1 Monitoring - BA015
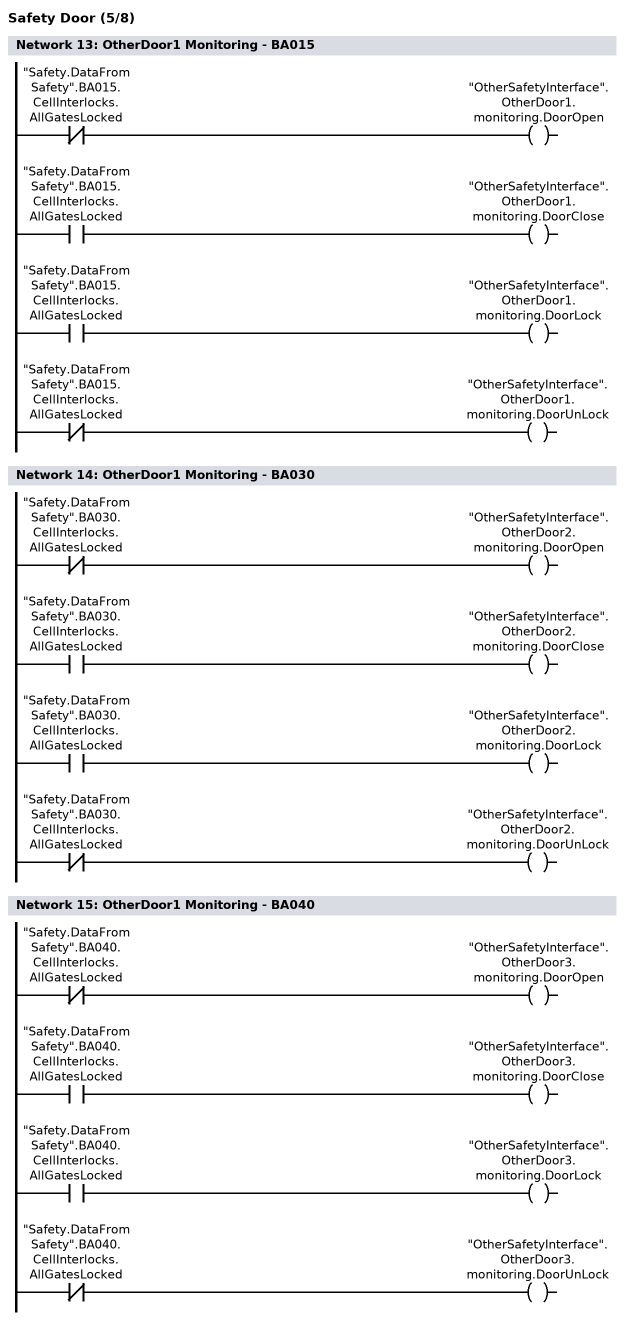
   RUNG wire#powerrail
      I_Contact( "Safety.DataFromSafety".BA015.CellInterlocks.AllGatesLocked )
      Coil( "OtherSafetyInterface".OtherDoor1.monitoring.DoorOpen )
   END_RUNG
   RUNG wire#powerrail
      Contact( "Safety.DataFromSafety".BA015.CellInterlocks.AllGatesLocked )
      Coil( "OtherSafetyInterface".OtherDoor1.monitoring.DoorClose )
   END_RUNG
   RUNG wire#powerrail
      Contact( "Safety.DataFromSafety".BA015.CellInterlocks.AllGatesLocked )
      Coil( "OtherSafetyInterface".OtherDoor1.monitoring.DoorLock )
   END_RUNG
   RUNG wire#powerrail
      I_Contact( "Safety.DataFromSafety".BA015.CellInterlocks.AllGatesLocked )
      Coil( "OtherSafetyInterface".OtherDoor1.monitoring.DoorUnLock )
   END_RUNG
   // the same network as SCL:
   "OtherSafetyInterface".OtherDoor1.monitoring.DoorOpen := NOT "Safety.DataFromSafety".BA015.CellInterlocks.AllGatesLocked;
   "OtherSafetyInterface".OtherDoor1.monitoring.DoorClose := "Safety.DataFromSafety".BA015.CellInterlocks.AllGatesLocked;
   "OtherSafetyInterface".OtherDoor1.monitoring.DoorLock := "Safety.DataFromSafety".BA015.CellInterlocks.AllGatesLocked;
   "OtherSafetyInterface".OtherDoor1.monitoring.DoorUnLock := NOT "Safety.DataFromSafety".BA015.CellInterlocks.AllGatesLocked;
END_REGION

REGION Network 14: OtherDoor1 Monitoring - BA030
   RUNG wire#powerrail
      I_Contact( "Safety.DataFromSafety".BA030.CellInterlocks.AllGatesLocked )
      Coil( "OtherSafetyInterface".OtherDoor2.monitoring.DoorOpen )
   END_RUNG
   RUNG wire#powerrail
      Contact( "Safety.DataFromSafety".BA030.CellInterlocks.AllGatesLocked )
      Coil( "OtherSafetyInterface".OtherDoor2.monitoring.DoorClose )
   END_RUNG
   RUNG wire#powerrail
      Contact( "Safety.DataFromSafety".BA030.CellInterlocks.AllGatesLocked )
      Coil( "OtherSafetyInterface".OtherDoor2.monitoring.DoorLock )
   END_RUNG
   RUNG wire#powerrail
      I_Contact( "Safety.DataFromSafety".BA030.CellInterlocks.AllGatesLocked )
      Coil( "OtherSafetyInterface".OtherDoor2.monitoring.DoorUnLock )
   END_RUNG
   // the same network as SCL:
   "OtherSafetyInterface".OtherDoor2.monitoring.DoorOpen := NOT "Safety.DataFromSafety".BA030.CellInterlocks.AllGatesLocked;
   "OtherSafetyInterface".OtherDoor2.monitoring.DoorClose := "Safety.DataFromSafety".BA030.CellInterlocks.AllGatesLocked;
   "OtherSafetyInterface".OtherDoor2.monitoring.DoorLock := "Safety.DataFromSafety".BA030.CellInterlocks.AllGatesLocked;
   "OtherSafetyInterface".OtherDoor2.monitoring.DoorUnLock := NOT "Safety.DataFromSafety".BA030.CellInterlocks.AllGatesLocked;
END_REGION

REGION Network 15: OtherDoor1 Monitoring - BA040
   RUNG wire#powerrail
      I_Contact( "Safety.DataFromSafety".BA040.CellInterlocks.AllGatesLocked )
      Coil( "OtherSafetyInterface".OtherDoor3.monitoring.DoorOpen )
   END_RUNG
   RUNG wire#powerrail
      Contact( "Safety.DataFromSafety".BA040.CellInterlocks.AllGatesLocked )
      Coil( "OtherSafetyInterface".OtherDoor3.monitoring.DoorClose )
   END_RUNG
   RUNG wire#powerrail
      Contact( "Safety.DataFromSafety".BA040.CellInterlocks.AllGatesLocked )
      Coil( "OtherSafetyInterface".OtherDoor3.monitoring.DoorLock )
   END_RUNG
   RUNG wire#powerrail
      I_Contact( "Safety.DataFromSafety".BA040.CellInterlocks.AllGatesLocked )
      Coil( "OtherSafetyInterface".OtherDoor3.monitoring.DoorUnLock )
   END_RUNG
   // the same network as SCL:
   "OtherSafetyInterface".OtherDoor3.monitoring.DoorOpen := NOT "Safety.DataFromSafety".BA040.CellInterlocks.AllGatesLocked;
   "OtherSafetyInterface".OtherDoor3.monitoring.DoorClose := "Safety.DataFromSafety".BA040.CellInterlocks.AllGatesLocked;
   "OtherSafetyInterface".OtherDoor3.monitoring.DoorLock := "Safety.DataFromSafety".BA040.CellInterlocks.AllGatesLocked;
   "OtherSafetyInterface".OtherDoor3.monitoring.DoorUnLock := NOT "Safety.DataFromSafety".BA040.CellInterlocks.AllGatesLocked;
END_REGION

REGION Network 16: OtherDoor1 Monitoring - BA060
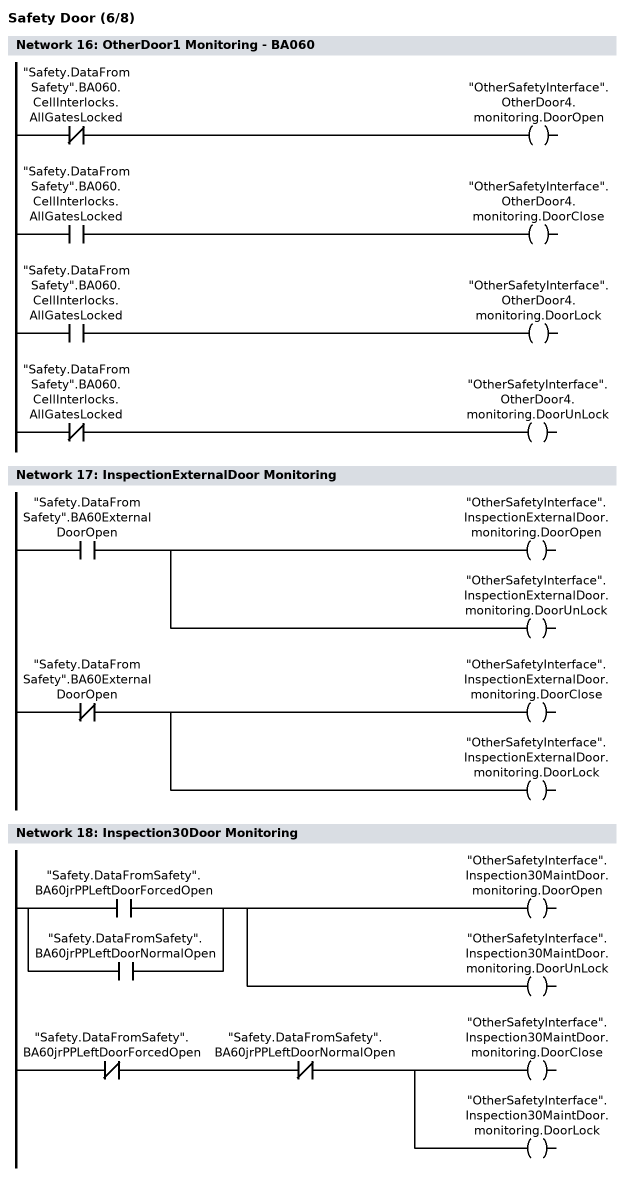
   RUNG wire#powerrail
      I_Contact( "Safety.DataFromSafety".BA060.CellInterlocks.AllGatesLocked )
      Coil( "OtherSafetyInterface".OtherDoor4.monitoring.DoorOpen )
   END_RUNG
   RUNG wire#powerrail
      Contact( "Safety.DataFromSafety".BA060.CellInterlocks.AllGatesLocked )
      Coil( "OtherSafetyInterface".OtherDoor4.monitoring.DoorClose )
   END_RUNG
   RUNG wire#powerrail
      Contact( "Safety.DataFromSafety".BA060.CellInterlocks.AllGatesLocked )
      Coil( "OtherSafetyInterface".OtherDoor4.monitoring.DoorLock )
   END_RUNG
   RUNG wire#powerrail
      I_Contact( "Safety.DataFromSafety".BA060.CellInterlocks.AllGatesLocked )
      Coil( "OtherSafetyInterface".OtherDoor4.monitoring.DoorUnLock )
   END_RUNG
   // the same network as SCL:
   "OtherSafetyInterface".OtherDoor4.monitoring.DoorOpen := NOT "Safety.DataFromSafety".BA060.CellInterlocks.AllGatesLocked;
   "OtherSafetyInterface".OtherDoor4.monitoring.DoorClose := "Safety.DataFromSafety".BA060.CellInterlocks.AllGatesLocked;
   "OtherSafetyInterface".OtherDoor4.monitoring.DoorLock := "Safety.DataFromSafety".BA060.CellInterlocks.AllGatesLocked;
   "OtherSafetyInterface".OtherDoor4.monitoring.DoorUnLock := NOT "Safety.DataFromSafety".BA060.CellInterlocks.AllGatesLocked;
END_REGION

REGION Network 17: InspectionExternalDoor Monitoring
   RUNG wire#powerrail
      Contact( "Safety.DataFromSafety".BA60ExternalDoorOpen )
      wire#w1
      Coil( "OtherSafetyInterface".InspectionExternalDoor.monitoring.DoorOpen )
   END_RUNG
   RUNG wire#w1
      Coil( "OtherSafetyInterface".InspectionExternalDoor.monitoring.DoorUnLock )
   END_RUNG
   RUNG wire#powerrail
      I_Contact( "Safety.DataFromSafety".BA60ExternalDoorOpen )
      wire#w2
      Coil( "OtherSafetyInterface".InspectionExternalDoor.monitoring.DoorClose )
   END_RUNG
   RUNG wire#w2
      Coil( "OtherSafetyInterface".InspectionExternalDoor.monitoring.DoorLock )
   END_RUNG
   // the same network as SCL:
   "OtherSafetyInterface".InspectionExternalDoor.monitoring.DoorOpen := "Safety.DataFromSafety".BA60ExternalDoorOpen;
   "OtherSafetyInterface".InspectionExternalDoor.monitoring.DoorUnLock := "Safety.DataFromSafety".BA60ExternalDoorOpen;
   "OtherSafetyInterface".InspectionExternalDoor.monitoring.DoorClose := NOT "Safety.DataFromSafety".BA60ExternalDoorOpen;
   "OtherSafetyInterface".InspectionExternalDoor.monitoring.DoorLock := NOT "Safety.DataFromSafety".BA60ExternalDoorOpen;
END_REGION

REGION Network 18: Inspection30Door Monitoring
   RUNG wire#powerrail
      Contact( "Safety.DataFromSafety".BA60jrPPLeftDoorForcedOpen )
      wire#w1
      Coil( "OtherSafetyInterface".Inspection30MaintDoor.monitoring.DoorOpen )
   END_RUNG
   RUNG wire#powerrail
      Contact( "Safety.DataFromSafety".BA60jrPPLeftDoorNormalOpen )
   END_RUNG wire#w1
   RUNG wire#w1
      Coil( "OtherSafetyInterface".Inspection30MaintDoor.monitoring.DoorUnLock )
   END_RUNG
   RUNG wire#powerrail
      I_Contact( "Safety.DataFromSafety".BA60jrPPLeftDoorForcedOpen )
      I_Contact( "Safety.DataFromSafety".BA60jrPPLeftDoorNormalOpen )
      wire#w2
      Coil( "OtherSafetyInterface".Inspection30MaintDoor.monitoring.DoorClose )
   END_RUNG
   RUNG wire#w2
      Coil( "OtherSafetyInterface".Inspection30MaintDoor.monitoring.DoorLock )
   END_RUNG
   // the same network as SCL:
   "OtherSafetyInterface".Inspection30MaintDoor.monitoring.DoorOpen := "Safety.DataFromSafety".BA60jrPPLeftDoorForcedOpen OR "Safety.DataFromSafety".BA60jrPPLeftDoorNormalOpen;
   "OtherSafetyInterface".Inspection30MaintDoor.monitoring.DoorUnLock := "OtherSafetyInterface".Inspection30MaintDoor.monitoring.DoorOpen;
   "OtherSafetyInterface".Inspection30MaintDoor.monitoring.DoorClose := NOT "Safety.DataFromSafety".BA60jrPPLeftDoorForcedOpen AND NOT "Safety.DataFromSafety".BA60jrPPLeftDoorNormalOpen;
   "OtherSafetyInterface".Inspection30MaintDoor.monitoring.DoorLock := "OtherSafetyInterface".Inspection30MaintDoor.monitoring.DoorClose;
END_REGION

REGION Network 19: Inspection40Door Monitoring
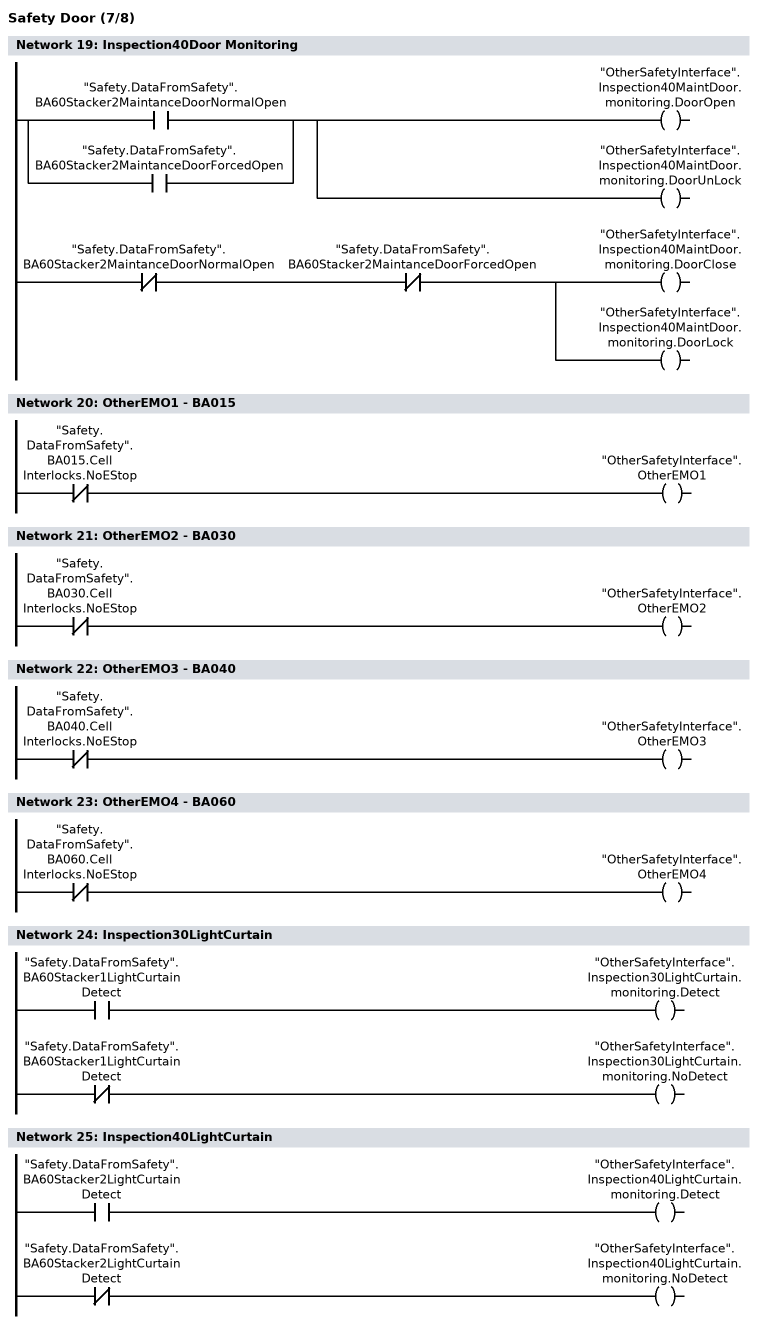
   RUNG wire#powerrail
      Contact( "Safety.DataFromSafety".BA60Stacker2MaintanceDoorNormalOpen )
      wire#w1
      Coil( "OtherSafetyInterface".Inspection40MaintDoor.monitoring.DoorOpen )
   END_RUNG
   RUNG wire#powerrail
      Contact( "Safety.DataFromSafety".BA60Stacker2MaintanceDoorForcedOpen )
   END_RUNG wire#w1
   RUNG wire#w1
      Coil( "OtherSafetyInterface".Inspection40MaintDoor.monitoring.DoorUnLock )
   END_RUNG
   RUNG wire#powerrail
      I_Contact( "Safety.DataFromSafety".BA60Stacker2MaintanceDoorNormalOpen )
      I_Contact( "Safety.DataFromSafety".BA60Stacker2MaintanceDoorForcedOpen )
      wire#w2
      Coil( "OtherSafetyInterface".Inspection40MaintDoor.monitoring.DoorClose )
   END_RUNG
   RUNG wire#w2
      Coil( "OtherSafetyInterface".Inspection40MaintDoor.monitoring.DoorLock )
   END_RUNG
   // the same network as SCL:
   "OtherSafetyInterface".Inspection40MaintDoor.monitoring.DoorOpen := "Safety.DataFromSafety".BA60Stacker2MaintanceDoorNormalOpen OR "Safety.DataFromSafety".BA60Stacker2MaintanceDoorForcedOpen;
   "OtherSafetyInterface".Inspection40MaintDoor.monitoring.DoorUnLock := "OtherSafetyInterface".Inspection40MaintDoor.monitoring.DoorOpen;
   "OtherSafetyInterface".Inspection40MaintDoor.monitoring.DoorClose := NOT "Safety.DataFromSafety".BA60Stacker2MaintanceDoorNormalOpen AND NOT "Safety.DataFromSafety".BA60Stacker2MaintanceDoorForcedOpen;
   "OtherSafetyInterface".Inspection40MaintDoor.monitoring.DoorLock := "OtherSafetyInterface".Inspection40MaintDoor.monitoring.DoorClose;
END_REGION

REGION Network 20: OtherEMO1 - BA015
   RUNG wire#powerrail
      I_Contact( "Safety.DataFromSafety".BA015.CellInterlocks.NoEStop )
      Coil( "OtherSafetyInterface".OtherEMO1 )
   END_RUNG
   // the same network as SCL:
   "OtherSafetyInterface".OtherEMO1 := NOT "Safety.DataFromSafety".BA015.CellInterlocks.NoEStop;
END_REGION

REGION Network 21: OtherEMO2 - BA030
   RUNG wire#powerrail
      I_Contact( "Safety.DataFromSafety".BA030.CellInterlocks.NoEStop )
      Coil( "OtherSafetyInterface".OtherEMO2 )
   END_RUNG
   // the same network as SCL:
   "OtherSafetyInterface".OtherEMO2 := NOT "Safety.DataFromSafety".BA030.CellInterlocks.NoEStop;
END_REGION

REGION Network 22: OtherEMO3 - BA040
   RUNG wire#powerrail
      I_Contact( "Safety.DataFromSafety".BA040.CellInterlocks.NoEStop )
      Coil( "OtherSafetyInterface".OtherEMO3 )
   END_RUNG
   // the same network as SCL:
   "OtherSafetyInterface".OtherEMO3 := NOT "Safety.DataFromSafety".BA040.CellInterlocks.NoEStop;
END_REGION

REGION Network 23: OtherEMO4 - BA060
   RUNG wire#powerrail
      I_Contact( "Safety.DataFromSafety".BA060.CellInterlocks.NoEStop )
      Coil( "OtherSafetyInterface".OtherEMO4 )
   END_RUNG
   // the same network as SCL:
   "OtherSafetyInterface".OtherEMO4 := NOT "Safety.DataFromSafety".BA060.CellInterlocks.NoEStop;
END_REGION

REGION Network 24: Inspection30LightCurtain
   RUNG wire#powerrail
      Contact( "Safety.DataFromSafety".BA60Stacker1LightCurtainDetect )
      Coil( "OtherSafetyInterface".Inspection30LightCurtain.monitoring.Detect )
   END_RUNG
   RUNG wire#powerrail
      I_Contact( "Safety.DataFromSafety".BA60Stacker1LightCurtainDetect )
      Coil( "OtherSafetyInterface".Inspection30LightCurtain.monitoring.NoDetect )
   END_RUNG
   // the same network as SCL:
   "OtherSafetyInterface".Inspection30LightCurtain.monitoring.Detect := "Safety.DataFromSafety".BA60Stacker1LightCurtainDetect;
   "OtherSafetyInterface".Inspection30LightCurtain.monitoring.NoDetect := NOT "Safety.DataFromSafety".BA60Stacker1LightCurtainDetect;
END_REGION

REGION Network 25: Inspection40LightCurtain
   RUNG wire#powerrail
      Contact( "Safety.DataFromSafety".BA60Stacker2LightCurtainDetect )
      Coil( "OtherSafetyInterface".Inspection40LightCurtain.monitoring.Detect )
   END_RUNG
   RUNG wire#powerrail
      I_Contact( "Safety.DataFromSafety".BA60Stacker2LightCurtainDetect )
      Coil( "OtherSafetyInterface".Inspection40LightCurtain.monitoring.NoDetect )
   END_RUNG
   // the same network as SCL:
   "OtherSafetyInterface".Inspection40LightCurtain.monitoring.Detect := "Safety.DataFromSafety".BA60Stacker2LightCurtainDetect;
   "OtherSafetyInterface".Inspection40LightCurtain.monitoring.NoDetect := NOT "Safety.DataFromSafety".BA60Stacker2LightCurtainDetect;
END_REGION

REGION Network 26: 30CathodeConveyorCover
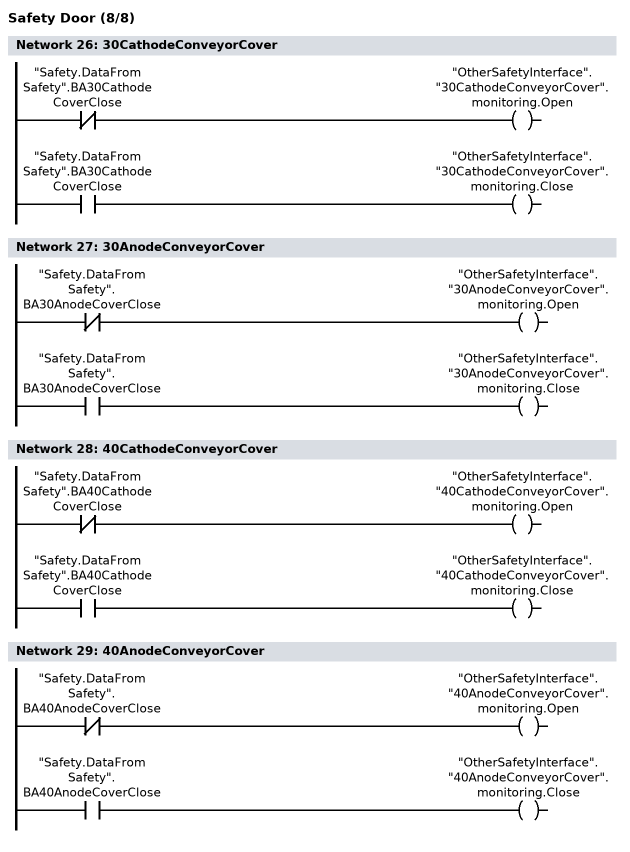
   RUNG wire#powerrail
      I_Contact( "Safety.DataFromSafety".BA30CathodeCoverClose )
      Coil( "OtherSafetyInterface"."30CathodeConveyorCover".monitoring.Open )
   END_RUNG
   RUNG wire#powerrail
      Contact( "Safety.DataFromSafety".BA30CathodeCoverClose )
      Coil( "OtherSafetyInterface"."30CathodeConveyorCover".monitoring.Close )
   END_RUNG
   // the same network as SCL:
   "OtherSafetyInterface"."30CathodeConveyorCover".monitoring.Open := NOT "Safety.DataFromSafety".BA30CathodeCoverClose;
   "OtherSafetyInterface"."30CathodeConveyorCover".monitoring.Close := "Safety.DataFromSafety".BA30CathodeCoverClose;
END_REGION

REGION Network 27: 30AnodeConveyorCover
   RUNG wire#powerrail
      I_Contact( "Safety.DataFromSafety".BA30AnodeCoverClose )
      Coil( "OtherSafetyInterface"."30AnodeConveyorCover".monitoring.Open )
   END_RUNG
   RUNG wire#powerrail
      Contact( "Safety.DataFromSafety".BA30AnodeCoverClose )
      Coil( "OtherSafetyInterface"."30AnodeConveyorCover".monitoring.Close )
   END_RUNG
   // the same network as SCL:
   "OtherSafetyInterface"."30AnodeConveyorCover".monitoring.Open := NOT "Safety.DataFromSafety".BA30AnodeCoverClose;
   "OtherSafetyInterface"."30AnodeConveyorCover".monitoring.Close := "Safety.DataFromSafety".BA30AnodeCoverClose;
END_REGION

REGION Network 28: 40CathodeConveyorCover
   RUNG wire#powerrail
      I_Contact( "Safety.DataFromSafety".BA40CathodeCoverClose )
      Coil( "OtherSafetyInterface"."40CathodeConveyorCover".monitoring.Open )
   END_RUNG
   RUNG wire#powerrail
      Contact( "Safety.DataFromSafety".BA40CathodeCoverClose )
      Coil( "OtherSafetyInterface"."40CathodeConveyorCover".monitoring.Close )
   END_RUNG
   // the same network as SCL:
   "OtherSafetyInterface"."40CathodeConveyorCover".monitoring.Open := NOT "Safety.DataFromSafety".BA40CathodeCoverClose;
   "OtherSafetyInterface"."40CathodeConveyorCover".monitoring.Close := "Safety.DataFromSafety".BA40CathodeCoverClose;
END_REGION

REGION Network 29: 40AnodeConveyorCover
   RUNG wire#powerrail
      I_Contact( "Safety.DataFromSafety".BA40AnodeCoverClose )
      Coil( "OtherSafetyInterface"."40AnodeConveyorCover".monitoring.Open )
   END_RUNG
   RUNG wire#powerrail
      Contact( "Safety.DataFromSafety".BA40AnodeCoverClose )
      Coil( "OtherSafetyInterface"."40AnodeConveyorCover".monitoring.Close )
   END_RUNG
   // the same network as SCL:
   "OtherSafetyInterface"."40AnodeConveyorCover".monitoring.Open := NOT "Safety.DataFromSafety".BA40AnodeCoverClose;
   "OtherSafetyInterface"."40AnodeConveyorCover".monitoring.Close := "Safety.DataFromSafety".BA40AnodeCoverClose;
END_REGION
END_FUNCTION

FUNCTION "CallProductionData" : Void   // FC151, LAD
TITLE = Produktions Daten / Production data
AUTHOR : SICAR
FAMILY : ProdData
VERSION : 1.0
// Dieser Baustein dient als Aufrufschnittstelle für die Funktionsbausteine  
// * _Shiftmodel  
// * _ProdDataCycleTimer  
// * _ProdDataCounter  
// * _ProdDataLimitValues  
// * _ProdDataShiftCounter  
// oder  
// * _ProdDataShiftCounterOee, ShiftProductionTimes
// Call of  FC ProductDataSimulation and LSicar Production Blocks
// stored: IsIECCheckEnabled true, SetENOAutomatically true
   // Ret_Val : Ret_Val
   VAR_TEMP   // added for the SCL form of the ladder/FBD networks
      _w1 : Bool;
      _w2 : Bool;
      _w3 : Bool;
      _w4 : Bool;
      _w5 : Bool;
      _w6 : Bool;
   END_VAR
BEGIN

REGION Network 1: BLOCK INFO HEADER
   // SIEMENS AG / (c)Copyright 2023
   // ------------------------------------------------------------------------------
   // Title:            CallProductionData(FC151)
   // Comment/Function: Call of  FC ProductDataSimulation and LSicar Production Blocks
   // Library/Family:   Automation Framework
   // Author:           Siemens Digital Industry
   // Tested with:      ---
   // Engineering:      TIA Portal V19
   // Restrictions:     -
   // Requirements:     ---
   // ------------------------------------------------------------------------------
   // Change log table:
   // Version  | Date       | Expert in charge       | Changes applied
   // ---------|------------|------------------------|------------------------------
   // 01.00.00 | 11.12.2023 | Siemens Industry Online Support
   //                         First released version
END_REGION

REGION Network 2: Beschreibung / DESCRIPTION
   // **Aufrufschnittstelle**  
   // Der Baustein wird einmalig im zyklischen Programm aufgerufen.  
   // 
   // 
   // #### Weitere Hinweise
   // 
   // #### Updateinfo
   // 
   // #### Weitere Dokumente
   // 
   // ![Icon](_Icon/reference.PNG)
   // 
   // Siehe:  
   // ..\Library Types\LSicar_Shiftmodel.pdf  
   // ..\Library Types\LSicar_ProdDataCycleTimer.pdf  
   // ..\Library Types\LSicar_ProdDataCounter.pdf  
   // ..\Library Types\LSicar_ProdDataLimitValues.pdf  
   // ..\Library Types\LSicar_ProdDataShiftCounter.pdf  
   // ..\Library Types\LSicar_ProdDataShiftCounterOee.pdf  
   // ..\Library Types\LSicar_ShiftProductionTimes.pdf
   // The block is used as a calling interface for the function blocks  
   // *   _Shiftmodel
   // *   _ProdDataCycleTimer
   // *   _ProdDataCounter
   // *   _ProdDataLimitValues
   // *   _ProdDataShiftCounter
   // or
   // *   _ProdDataShiftCounterOee, ShiftProductionTimes
   // 
   // **Calling interface**  
   // The block must be called once only in the cyclic program.  
   // 
   // The block is used as a calling interface for the function blocks  
   // *   _Shiftmodel
   // *   _ProdDataCycleTimer
   // *   _ProdDataCounter
   // *   _ProdDataLimitValues
   // *   _ProdDataShiftCounter
   // or
   // *   _ProdDataShiftCounterOee, ShiftProductionTimes
   // 
   // #### Additional information
   // 
   // #### Update info
   // 
   // #### Further documentations
   // 
   // ![Icon](_Icon/reference.PNG) 
   // 
   // See:  
   // ..\Library Types\LSicar_Shiftmodel.pdf  
   // ..\Library Types\LSicar_ProdDataCycleTimer.pdf  
   // ..\Library Types\LSicar_ProdDataCounter.pdf  
   // ..\Library Types\LSicar_ProdDataLimitValues.pdf  
   // ..\Library Types\LSicar_ProdDataShiftCounter.pdf  
   // ..\Library Types\LSicar_ProdDataShiftCounterOee.pdf  
   // ..\Library Types\LSicar_ShiftProductionTimes.pdf
END_REGION

REGION Network 3: Beispiel: Counter 1..2 / Call production data counter
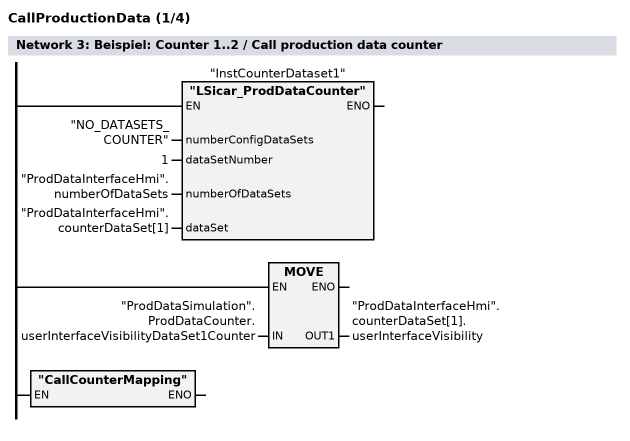
   RUNG wire#powerrail
      "InstCounterDataset1"(numberConfigDataSets := "NO_DATASETS_COUNTER", dataSetNumber := 1, numberOfDataSets := "ProdDataInterfaceHmi".numberOfDataSets, dataSet := "ProdDataInterfaceHmi".counterDataSet[1])
   END_RUNG
   RUNG wire#powerrail
      Move(in := "ProdDataSimulation".ProdDataCounter.userInterfaceVisibilityDataSet1Counter, out1 => "ProdDataInterfaceHmi".counterDataSet[1].userInterfaceVisibility)
   END_RUNG
   RUNG wire#powerrail
      "CallCounterMapping"()
   END_RUNG
   // the same network as SCL:
   "InstCounterDataset1"(numberConfigDataSets := "NO_DATASETS_COUNTER",   // "LSicar_ProdDataCounter"
                         dataSetNumber := 1,
                         numberOfDataSets := "ProdDataInterfaceHmi".numberOfDataSets,
                         dataSet := "ProdDataInterfaceHmi".counterDataSet[1]);
   "ProdDataInterfaceHmi".counterDataSet[1].userInterfaceVisibility := "ProdDataSimulation".ProdDataCounter.userInterfaceVisibilityDataSet1Counter;
   "CallCounterMapping"();
END_REGION

